LIN {X 0,Y 566.722,Z 306.411,A -85,B 0,C 180,E1 -2622.534,E2 -2622.534} C_VEL
LIN {X 0,Y 565.899,Z 301.524,A -85,B 0,C 180,E1 -2622.643,E2 -2622.643} C_VEL
LIN {X 0,Y 565.948,Z 295.461,A -85,B 0,C 180,E1 -2625.116,E2 -2625.116} C_VEL
LIN {X 0,Y 565.984,Z 288.275,A -85,B 0,C 180,E1 -2628.085,E2 -2628.085} C_VEL
LIN {X 0,Y 566.059,Z 281.089,A -85,B 0,C 180,E1 -2631.103,E2 -2631.103} C_VEL
LIN {X 0,Y 566.08,Z 273.903,A -85,B 0,C 180,E1 -2634.186,E2 -2634.186} C_VEL
LIN {X 0,Y 566.13,Z 268.296,A -85,B 0,C 180,E1 -2636.641,E2 -2636.641} C_VEL
LIN {X 0,Y 566.201,Z 261.327,A -85,B 0,C 180,E1 -2639.768,E2 -2639.768} C_VEL
LIN {X 0,Y 566.246,Z 255.555,A -85,B 0,C 180,E1 -2642.434,E2 -2642.434} C_VEL
LIN {X 0,Y 566.295,Z 250.149,A -85,B 0,C 180,E1 -2645.004,E2 -2645.004} C_VEL
LIN {X 0,Y 566.408,Z 245.469,A -85,B 0,C 180,E1 -2647.444,E2 -2647.444} C_VEL
LIN {X 0,Y 566.539,Z 240.518,A -85,B 0,C 180,E1 -2650.17,E2 -2650.17} C_VEL
LIN {X 0,Y 566.466,Z 237.367,A -85,B 0,C 180,E1 -2652.063,E2 -2652.063} C_VEL
LIN {X 0,Y 566.201,Z 235.83,A -85,B 0,C 180,E1 -2653.053,E2 -2653.053} C_VEL
LIN {X 0,Y 566.162,Z 235.462,A -85,B 0,C 180,E1 -2654.038,E2 -2654.038} C_VEL
LIN {X 0,Y 566.185,Z 235.462,A -85,B 0,C 180,E1 -2657.083,E2 -2657.083} C_VEL
LIN {X 0,Y 566.209,Z 235.454,A -85,B 0,C 180,E1 -2660.314,E2 -2660.314} C_VEL
LIN {X 0,Y 566.182,Z 235.455,A -85,B 0,C 180,E1 -2663.426,E2 -2663.426} C_VEL
LIN {X 0,Y 566.199,Z 235.455,A -85,B 0,C 180,E1 -2666.266,E2 -2666.266} C_VEL
LIN {X 0,Y 566.186,Z 235.458,A -85,B 0,C 180,E1 -2668.923,E2 -2668.923} C_VEL
LIN {X 0,Y 566.15,Z 235.459,A -85,B 0,C 180,E1 -2671.851,E2 -2671.851} C_VEL
LIN {X 0,Y 566.193,Z 235.458,A -85,B 0,C 180,E1 -2674.247,E2 -2674.247} C_VEL
LIN {X 0,Y 566.161,Z 235.456,A -85,B 0,C 180,E1 -2677.365,E2 -2677.365} C_VEL
LIN {X 0,Y 566.17,Z 235.456,A -85,B 0,C 180,E1 -2679.658,E2 -2679.658} C_VEL
LIN {X 0,Y 566.166,Z 235.46,A -85,B 0,C 180,E1 -2681.917,E2 -2681.917} C_VEL
LIN {X 0,Y 566.182,Z 235.454,A -85,B 0,C 180,E1 -2684.887,E2 -2684.887} C_VEL
LIN {X 0,Y 566.21,Z 235.456,A -85,B 0,C 180,E1 -2687.815,E2 -2687.815} C_VEL
LIN {X 0,Y 566.16,Z 235.466,A -85,B 0,C 180,E1 -2689.988,E2 -2689.988} C_VEL
LIN {X 0,Y 566.185,Z 235.459,A -85,B 0,C 180,E1 -2692.149,E2 -2692.149} C_VEL
LIN {X 0,Y 566.256,Z 235.445,A -85,B 0,C 180,E1 -2695.012,E2 -2695.012} C_VEL
LIN {X 0,Y 566.262,Z 235.451,A -85,B 0,C 180,E1 -2697.862,E2 -2697.862} C_VEL
LIN {X 0,Y 566.269,Z 235.447,A -85,B 0,C 180,E1 -2699.996,E2 -2699.996} C_VEL
LIN {X 0,Y 566.244,Z 235.446,A -85,B 0,C 180,E1 -2702.841,E2 -2702.841} C_VEL
LIN {X 0,Y 566.236,Z 235.454,A -85,B 0,C 180,E1 -2705.694,E2 -2705.694} C_VEL
LIN {X 0,Y 566.177,Z 235.454,A -85,B 0,C 180,E1 -2708.562,E2 -2708.562} C_VEL
LIN {X 0,Y 566.226,Z 235.456,A -85,B 0,C 180,E1 -2711.45,E2 -2711.45} C_VEL
LIN {X 0,Y 566.184,Z 235.454,A -85,B 0,C 180,E1 -2714.49,E2 -2714.49} C_VEL
LIN {X 0,Y 566.173,Z 235.462,A -85,B 0,C 180,E1 -2717.327,E2 -2717.327} C_VEL
LIN {X 0,Y 566.179,Z 235.454,A -85,B 0,C 180,E1 -2720.333,E2 -2720.333} C_VEL
LIN {X 0,Y 566.141,Z 235.464,A -85,B 0,C 180,E1 -2723.277,E2 -2723.277} C_VEL
LIN {X 0,Y 566.176,Z 235.454,A -85,B 0,C 180,E1 -2725.745,E2 -2725.745} C_VEL
LIN {X 0,Y 566.174,Z 235.456,A -85,B 0,C 180,E1 -2727.443,E2 -2727.443} C_VEL
LIN {X 0,Y 565.499,Z 235.54,A -85,B 0,C 180,E1 -2728.037,E2 -2728.037} C_VEL
LIN {X 0,Y 562.633,Z 235.902,A -85,B 0,C 180,E1 -2729.001,E2 -2729.001} C_VEL
LIN {X 0,Y 560.217,Z 236.2,A -85,B 0,C 180,E1 -2729.776,E2 -2729.776} C_VEL
LIN {X 0,Y 559.185,Z 236.329,A -85,B 0,C 180,E1 -2730.375,E2 -2730.375} C_VEL
LIN {X 0,Y 559.103,Z 236.337,A -85,B 0,C 180,E1 -2730.578,E2 -2730.578} C_VEL
LIN {X 0,Y 559.116,Z 236.344,A -85,B 0,C 180,E1 -2732.711,E2 -2732.711} C_VEL
LIN {X 0,Y 559.118,Z 236.334,A -85,B 0,C 180,E1 -2735.317,E2 -2735.317} C_VEL
LIN {X 0,Y 559.09,Z 236.339,A -85,B 0,C 180,E1 -2738.013,E2 -2738.013} C_VEL
LIN {X 0,Y 559.13,Z 236.336,A -85,B 0,C 180,E1 -2740.806,E2 -2740.806} C_VEL
LIN {X 0,Y 559.116,Z 236.335,A -85,B 0,C 180,E1 -2743.727,E2 -2743.727} C_VEL
LIN {X 0,Y 559.115,Z 236.336,A -85,B 0,C 180,E1 -2746.797,E2 -2746.797} C_VEL
LIN {X 0,Y 559.127,Z 236.332,A -85,B 0,C 180,E1 -2749.186,E2 -2749.186} C_VEL
LIN {X 0,Y 559.082,Z 236.345,A -85,B 0,C 180,E1 -2751.979,E2 -2751.979} C_VEL
LIN {X 0,Y 559.103,Z 236.336,A -85,B 0,C 180,E1 -2754.779,E2 -2754.779} C_VEL
LIN {X 0,Y 559.117,Z 236.335,A -85,B 0,C 180,E1 -2757.358,E2 -2757.358} C_VEL
LIN {X 0,Y 559.139,Z 236.337,A -85,B 0,C 180,E1 -2760.13,E2 -2760.13} C_VEL
LIN {X 0,Y 559.121,Z 236.334,A -85,B 0,C 180,E1 -2763.167,E2 -2763.167} C_VEL
LIN {X 0,Y 559.111,Z 236.34,A -85,B 0,C 180,E1 -2765.493,E2 -2765.493} C_VEL
LIN {X 0,Y 559.104,Z 236.342,A -85,B 0,C 180,E1 -2767.846,E2 -2767.846} C_VEL
LIN {X 0,Y 559.131,Z 236.332,A -85,B 0,C 180,E1 -2770.49,E2 -2770.49} C_VEL
LIN {X 0,Y 559.147,Z 236.336,A -85,B 0,C 180,E1 -2773.197,E2 -2773.197} C_VEL
LIN {X 0,Y 559.122,Z 236.335,A -85,B 0,C 180,E1 -2776.183,E2 -2776.183} C_VEL
LIN {X 0,Y 559.171,Z 236.334,A -85,B 0,C 180,E1 -2779.133,E2 -2779.133} C_VEL
LIN {X 0,Y 559.15,Z 236.331,A -85,B 0,C 180,E1 -2782.053,E2 -2782.053} C_VEL
LIN {X 0,Y 559.203,Z 236.33,A -85,B 0,C 180,E1 -2784.953,E2 -2784.953} C_VEL
LIN {X 0,Y 559.183,Z 236.327,A -85,B 0,C 180,E1 -2787.839,E2 -2787.839} C_VEL
LIN {X 0,Y 559.219,Z 236.328,A -85,B 0,C 180,E1 -2790.72,E2 -2790.72} C_VEL
LIN {X 0,Y 559.188,Z 236.334,A -85,B 0,C 180,E1 -2792.882,E2 -2792.882} C_VEL
LIN {X 0,Y 559.172,Z 236.328,A -85,B 0,C 180,E1 -2795.771,E2 -2795.771} C_VEL
LIN {X 0,Y 559.15,Z 236.331,A -85,B 0,C 180,E1 -2797.947,E2 -2797.947} C_VEL
LIN {X 0,Y 559.171,Z 236.334,A -85,B 0,C 180,E1 -2800.867,E2 -2800.867} C_VEL
LIN {X 0,Y 559.122,Z 236.335,A -85,B 0,C 180,E1 -2803.817,E2 -2803.817} C_VEL
LIN {X 0,Y 559.147,Z 236.336,A -85,B 0,C 180,E1 -2806.803,E2 -2806.803} C_VEL
LIN {X 0,Y 559.113,Z 236.336,A -85,B 0,C 180,E1 -2809.839,E2 -2809.839} C_VEL
LIN {X 0,Y 559.104,Z 236.342,A -85,B 0,C 180,E1 -2812.154,E2 -2812.154} C_VEL
LIN {X 0,Y 559.111,Z 236.34,A -85,B 0,C 180,E1 -2814.507,E2 -2814.507} C_VEL
LIN {X 0,Y 559.118,Z 236.334,A -85,B 0,C 180,E1 -2816.904,E2 -2816.904} C_VEL
LIN {X 0,Y 559.139,Z 236.337,A -85,B 0,C 180,E1 -2819.87,E2 -2819.87} C_VEL
LIN {X 0,Y 559.118,Z 236.334,A -85,B 0,C 180,E1 -2822.717,E2 -2822.717} C_VEL
LIN {X 0,Y 559.102,Z 236.337,A -85,B 0,C 180,E1 -2825.325,E2 -2825.325} C_VEL
LIN {X 0,Y 559.082,Z 236.345,A -85,B 0,C 180,E1 -2828.021,E2 -2828.021} C_VEL
LIN {X 0,Y 559.127,Z 236.332,A -85,B 0,C 180,E1 -2830.814,E2 -2830.814} C_VEL
LIN {X 0,Y 559.111,Z 236.343,A -85,B 0,C 180,E1 -2833.736,E2 -2833.736} C_VEL
LIN {X 0,Y 559.126,Z 236.333,A -85,B 0,C 180,E1 -2836.805,E2 -2836.805} C_VEL
LIN {X 0,Y 559.13,Z 236.336,A -85,B 0,C 180,E1 -2839.194,E2 -2839.194} C_VEL
LIN {X 0,Y 559.09,Z 236.339,A -85,B 0,C 180,E1 -2841.987,E2 -2841.987} C_VEL
LIN {X 0,Y 559.119,Z 236.335,A -85,B 0,C 180,E1 -2844.788,E2 -2844.788} C_VEL
LIN {X 0,Y 559.117,Z 236.342,A -85,B 0,C 180,E1 -2847.369,E2 -2847.369} C_VEL
LIN {X 0,Y 559.113,Z 236.334,A -85,B 0,C 180,E1 -2850.147,E2 -2850.147} C_VEL
LIN {X 0,Y 559.138,Z 236.341,A -85,B 0,C 180,E1 -2853.103,E2 -2853.103} C_VEL
LIN {X 0,Y 559.124,Z 236.336,A -85,B 0,C 180,E1 -2855.5,E2 -2855.5} C_VEL
LIN {X 0,Y 559.144,Z 236.335,A -85,B 0,C 180,E1 -2858.629,E2 -2858.629} C_VEL
LIN {X 0,Y 559.134,Z 236.34,A -85,B 0,C 180,E1 -2860.931,E2 -2860.931} C_VEL
LIN {X 0,Y 559.137,Z 236.331,A -85,B 0,C 180,E1 -2863.952,E2 -2863.952} C_VEL
LIN {X 0,Y 559.133,Z 236.338,A -85,B 0,C 180,E1 -2866.929,E2 -2866.929} C_VEL
LIN {X 0,Y 559.177,Z 236.329,A -85,B 0,C 180,E1 -2869.138,E2 -2869.138} C_VEL
LIN {X 0,Y 559.173,Z 236.329,A -85,B 0,C 180,E1 -2872.058,E2 -2872.058} C_VEL
LIN {X 0,Y 559.226,Z 236.323,A -85,B 0,C 180,E1 -2874.958,E2 -2874.958} C_VEL
LIN {X 0,Y 559.228,Z 236.322,A -85,B 0,C 180,E1 -2877.844,E2 -2877.844} C_VEL
LIN {X 0,Y 559.259,Z 236.319,A -85,B 0,C 180,E1 -2880.724,E2 -2880.724} C_VEL
LIN {X 0,Y 559.213,Z 236.323,A -85,B 0,C 180,E1 -2882.886,E2 -2882.886} C_VEL
LIN {X 0,Y 559.198,Z 236.327,A -85,B 0,C 180,E1 -2885.774,E2 -2885.774} C_VEL
LIN {X 0,Y 559.157,Z 236.33,A -85,B 0,C 180,E1 -2888.679,E2 -2888.679} C_VEL
LIN {X 0,Y 559.198,Z 236.327,A -85,B 0,C 180,E1 -2891.604,E2 -2891.604} C_VEL
LIN {X 0,Y 559.18,Z 236.327,A -85,B 0,C 180,E1 -2894.591,E2 -2894.591} C_VEL
LIN {X 0,Y 559.11,Z 236.34,A -85,B 0,C 180,E1 -2897.562,E2 -2897.562} C_VEL
LIN {X 0,Y 559.154,Z 236.337,A -85,B 0,C 180,E1 -2899.841,E2 -2899.841} C_VEL
LIN {X 0,Y 559.13,Z 236.334,A -85,B 0,C 180,E1 -2902.156,E2 -2902.156} C_VEL
LIN {X 0,Y 559.141,Z 236.334,A -85,B 0,C 180,E1 -2905.181,E2 -2905.181} C_VEL
LIN {X 0,Y 559.106,Z 236.341,A -85,B 0,C 180,E1 -2907.719,E2 -2907.719} C_VEL
LIN {X 0,Y 559.137,Z 236.332,A -85,B 0,C 180,E1 -2910.187,E2 -2910.187} C_VEL
LIN {X 0,Y 559.15,Z 236.331,A -85,B 0,C 180,E1 -2912.718,E2 -2912.718} C_VEL
LIN {X 0,Y 559.12,Z 236.342,A -85,B 0,C 180,E1 -2915.327,E2 -2915.327} C_VEL
LIN {X 0,Y 559.127,Z 236.334,A -85,B 0,C 180,E1 -2918.021,E2 -2918.021} C_VEL
LIN {X 0,Y 559.157,Z 236.336,A -85,B 0,C 180,E1 -2920.815,E2 -2920.815} C_VEL
LIN {X 0,Y 559.111,Z 236.339,A -85,B 0,C 180,E1 -2923.739,E2 -2923.739} C_VEL
LIN {X 0,Y 559.119,Z 236.342,A -85,B 0,C 180,E1 -2926.265,E2 -2926.265} C_VEL
LIN {X 0,Y 559.534,Z 239.189,A -85,B 0,C 180,E1 -2928.265,E2 -2928.265} C_VEL
LIN {X 0,Y 559.517,Z 242.348,A -85,B 0,C 180,E1 -2930.164,E2 -2930.164} C_VEL
LIN {X 0,Y 559.377,Z 247.292,A -85,B 0,C 180,E1 -2932.911,E2 -2932.911} C_VEL
LIN {X 0,Y 559.249,Z 252.345,A -85,B 0,C 180,E1 -2935.563,E2 -2935.563} C_VEL
LIN {X 0,Y 559.202,Z 257.734,A -85,B 0,C 180,E1 -2938.14,E2 -2938.14} C_VEL
LIN {X 0,Y 559.128,Z 263.124,A -85,B 0,C 180,E1 -2940.646,E2 -2940.646} C_VEL
LIN {X 0,Y 559.095,Z 268.727,A -85,B 0,C 180,E1 -2943.19,E2 -2943.19} C_VEL
LIN {X 0,Y 559.025,Z 273.903,A -85,B 0,C 180,E1 -2945.489,E2 -2945.489} C_VEL
LIN {X 0,Y 559.001,Z 281.089,A -85,B 0,C 180,E1 -2948.617,E2 -2948.617} C_VEL
LIN {X 0,Y 558.931,Z 286.478,A -85,B 0,C 180,E1 -2950.918,E2 -2950.918} C_VEL
LIN {X 0,Y 558.884,Z 291.868,A -85,B 0,C 180,E1 -2953.189,E2 -2953.189} C_VEL
LIN {X 0,Y 558.843,Z 299.054,A -85,B 0,C 180,E1 -2956.176,E2 -2956.176} C_VEL
LIN {X 0,Y 558.835,Z 301.524,A -85,B 0,C 180,E1 -2957.194,E2 -2957.194} C_VEL
LIN {X 0,Y 559.967,Z 309.414,A -85,B 0,C 180,E1 -2957.382,E2 -2957.382} C_VEL
LIN {X 0,Y 559.851,Z 321.119,A -85,B 0,C 180,E1 -2957.724,E2 -2957.724} C_VEL
LIN {X 0,Y 559.715,Z 331.464,A -85,B 0,C 180,E1 -2958.135,E2 -2958.135} C_VEL
LIN {X 0,Y 559.551,Z 342.846,A -85,B 0,C 180,E1 -2958.72,E2 -2958.72} C_VEL
LIN {X 0,Y 559.433,Z 354.75,A -85,B 0,C 180,E1 -2959.505,E2 -2959.505} C_VEL
LIN {X 0,Y 559.296,Z 363.641,A -85,B 0,C 180,E1 -2960.233,E2 -2960.233} C_VEL
LIN {X 0,Y 559.133,Z 372.762,A -85,B 0,C 180,E1 -2961.143,E2 -2961.143} C_VEL
LIN {X 0,Y 559.055,Z 380.309,A -85,B 0,C 180,E1 -2962.052,E2 -2962.052} C_VEL
LIN {X 0,Y 558.927,Z 387.956,A -85,B 0,C 180,E1 -2963.176,E2 -2963.176} C_VEL
LIN {X 0,Y 558.929,Z 393.682,A -85,B 0,C 180,E1 -2964.227,E2 -2964.227} C_VEL
LIN {X 0,Y 558.827,Z 398.379,A -85,B 0,C 180,E1 -2965.311,E2 -2965.311} C_VEL
LIN {X 0,Y 558.837,Z 401.966,A -85,B 0,C 180,E1 -2966.395,E2 -2966.395} C_VEL
LIN {X 0,Y 558.8,Z 403.792,A -85,B 0,C 180,E1 -2967.116,E2 -2967.116} C_VEL
LIN {X 0,Y 558.745,Z 406.19,A -85,B 0,C 180,E1 -2968.559,E2 -2968.559} C_VEL
LIN {X 0,Y 558.741,Z 406.782,A -85,B 0,C 180,E1 -2969.279,E2 -2969.279} C_VEL
LIN {X 0,Y 558.741,Z 406.782,A -85,B 0,C 180,E1 -2970.721,E2 -2970.721} C_VEL
LIN {X 0,Y 558.745,Z 406.19,A -85,B 0,C 180,E1 -2971.441,E2 -2971.441} C_VEL
LIN {X 0,Y 558.8,Z 403.792,A -85,B 0,C 180,E1 -2972.884,E2 -2972.884} C_VEL
LIN {X 0,Y 558.845,Z 400.88,A -85,B 0,C 180,E1 -2973.966,E2 -2973.966} C_VEL
LIN {X 0,Y 558.798,Z 396.93,A -85,B 0,C 180,E1 -2975.051,E2 -2975.051} C_VEL
LIN {X 0,Y 558.911,Z 391.835,A -85,B 0,C 180,E1 -2976.136,E2 -2976.136} C_VEL
LIN {X 0,Y 558.977,Z 385.452,A -85,B 0,C 180,E1 -2977.223,E2 -2977.223} C_VEL
LIN {X 0,Y 559.098,Z 377.491,A -85,B 0,C 180,E1 -2978.312,E2 -2978.312} C_VEL
LIN {X 0,Y 559.183,Z 369.35,A -85,B 0,C 180,E1 -2979.221,E2 -2979.221} C_VEL
LIN {X 0,Y 559.336,Z 359.358,A -85,B 0,C 180,E1 -2980.131,E2 -2980.131} C_VEL
LIN {X 0,Y 559.46,Z 349.539,A -85,B 0,C 180,E1 -2980.861,E2 -2980.861} C_VEL
LIN {X 0,Y 559.612,Z 338.508,A -85,B 0,C 180,E1 -2981.523,E2 -2981.523} C_VEL
LIN {X 0,Y 559.811,Z 324.985,A -85,B 0,C 180,E1 -2982.139,E2 -2982.139} C_VEL
LIN {X 0,Y 559.957,Z 312.983,A -85,B 0,C 180,E1 -2982.527,E2 -2982.527} C_VEL
LIN {X 0,Y 559.764,Z 307.128,A -85,B 0,C 180,E1 -2982.678,E2 -2982.678} C_VEL
LIN {X 0,Y 558.835,Z 301.524,A -85,B 0,C 180,E1 -2982.806,E2 -2982.806} C_VEL
LIN {X 0,Y 558.862,Z 295.461,A -85,B 0,C 180,E1 -2985.312,E2 -2985.312} C_VEL
LIN {X 0,Y 558.904,Z 288.275,A -85,B 0,C 180,E1 -2988.322,E2 -2988.322} C_VEL
LIN {X 0,Y 558.949,Z 282.885,A -85,B 0,C 180,E1 -2990.613,E2 -2990.613} C_VEL
LIN {X 0,Y 559.027,Z 276.436,A -85,B 0,C 180,E1 -2993.399,E2 -2993.399} C_VEL
LIN {X 0,Y 559.071,Z 270.31,A -85,B 0,C 180,E1 -2996.102,E2 -2996.102} C_VEL
LIN {X 0,Y 559.115,Z 264.92,A -85,B 0,C 180,E1 -2998.532,E2 -2998.532} C_VEL
LIN {X 0,Y 559.185,Z 258.975,A -85,B 0,C 180,E1 -3001.277,E2 -3001.277} C_VEL
LIN {X 0,Y 559.253,Z 253.328,A -85,B 0,C 180,E1 -3003.96,E2 -3003.96} C_VEL
LIN {X 0,Y 559.359,Z 248.434,A -85,B 0,C 180,E1 -3006.472,E2 -3006.472} C_VEL
LIN {X 0,Y 559.482,Z 243.98,A -85,B 0,C 180,E1 -3008.908,E2 -3008.908} C_VEL
LIN {X 0,Y 559.591,Z 240.185,A -85,B 0,C 180,E1 -3011.099,E2 -3011.099} C_VEL
LIN {X 0,Y 559.181,Z 236.927,A -85,B 0,C 180,E1 -3013.198,E2 -3013.198} C_VEL
LIN {X 0,Y 559.115,Z 236.341,A -85,B 0,C 180,E1 -3013.735,E2 -3013.735} C_VEL
LIN {X 0,Y 559.111,Z 236.338,A -85,B 0,C 180,E1 -3016.261,E2 -3016.261} C_VEL
LIN {X 0,Y 559.119,Z 236.34,A -85,B 0,C 180,E1 -3019.182,E2 -3019.182} C_VEL
LIN {X 0,Y 559.171,Z 236.333,A -85,B 0,C 180,E1 -3021.191,E2 -3021.191} C_VEL
LIN {X 0,Y 559.12,Z 236.333,A -85,B 0,C 180,E1 -3023.785,E2 -3023.785} C_VEL
LIN {X 0,Y 559.148,Z 236.335,A -85,B 0,C 180,E1 -3026.421,E2 -3026.421} C_VEL
LIN {X 0,Y 559.151,Z 236.333,A -85,B 0,C 180,E1 -3028.978,E2 -3028.978} C_VEL
LIN {X 0,Y 559.112,Z 236.334,A -85,B 0,C 180,E1 -3031.628,E2 -3031.628} C_VEL
LIN {X 0,Y 559.13,Z 236.337,A -85,B 0,C 180,E1 -3034.697,E2 -3034.697} C_VEL
LIN {X 0,Y 559.112,Z 236.335,A -85,B 0,C 180,E1 -3037.063,E2 -3037.063} C_VEL
LIN {X 0,Y 559.149,Z 236.33,A -85,B 0,C 180,E1 -3039.391,E2 -3039.391} C_VEL
LIN {X 0,Y 559.116,Z 236.336,A -85,B 0,C 180,E1 -3041.681,E2 -3041.681} C_VEL
LIN {X 0,Y 559.13,Z 236.334,A -85,B 0,C 180,E1 -3044.691,E2 -3044.691} C_VEL
LIN {X 0,Y 559.169,Z 236.331,A -85,B 0,C 180,E1 -3047.659,E2 -3047.659} C_VEL
LIN {X 0,Y 559.122,Z 236.341,A -85,B 0,C 180,E1 -3049.861,E2 -3049.861} C_VEL
LIN {X 0,Y 559.138,Z 236.339,A -85,B 0,C 180,E1 -3052.049,E2 -3052.049} C_VEL
LIN {X 0,Y 559.23,Z 236.32,A -85,B 0,C 180,E1 -3054.949,E2 -3054.949} C_VEL
LIN {X 0,Y 559.234,Z 236.327,A -85,B 0,C 180,E1 -3057.835,E2 -3057.835} C_VEL
LIN {X 0,Y 559.238,Z 236.323,A -85,B 0,C 180,E1 -3059.996,E2 -3059.996} C_VEL
LIN {X 0,Y 559.212,Z 236.322,A -85,B 0,C 180,E1 -3062.877,E2 -3062.877} C_VEL
LIN {X 0,Y 559.203,Z 236.328,A -85,B 0,C 180,E1 -3065.766,E2 -3065.766} C_VEL
LIN {X 0,Y 559.143,Z 236.331,A -85,B 0,C 180,E1 -3068.67,E2 -3068.67} C_VEL
LIN {X 0,Y 559.187,Z 236.33,A -85,B 0,C 180,E1 -3071.596,E2 -3071.596} C_VEL
LIN {X 0,Y 559.133,Z 236.333,A -85,B 0,C 180,E1 -3074.573,E2 -3074.573} C_VEL
LIN {X 0,Y 559.147,Z 236.339,A -85,B 0,C 180,E1 -3077.208,E2 -3077.208} C_VEL
LIN {X 0,Y 559.139,Z 236.332,A -85,B 0,C 180,E1 -3079.833,E2 -3079.833} C_VEL
LIN {X 0,Y 559.112,Z 236.334,A -85,B 0,C 180,E1 -3082.148,E2 -3082.148} C_VEL
LIN {X 0,Y 559.144,Z 236.334,A -85,B 0,C 180,E1 -3085.293,E2 -3085.293} C_VEL
LIN {X 0,Y 559.155,Z 236.329,A -85,B 0,C 180,E1 -3087.707,E2 -3087.707} C_VEL
LIN {X 0,Y 559.103,Z 236.337,A -85,B 0,C 180,E1 -3090.578,E2 -3090.578} C_VEL
LIN {X 0,Y 558.439,Z 236.423,A -85,B 0,C 180,E1 -3091.179,E2 -3091.179} C_VEL
LIN {X 0,Y 555.575,Z 236.777,A -85,B 0,C 180,E1 -3092.155,E2 -3092.155} C_VEL
LIN {X 0,Y 553.164,Z 237.081,A -85,B 0,C 180,E1 -3092.941,E2 -3092.941} C_VEL
LIN {X 0,Y 552.145,Z 237.203,A -85,B 0,C 180,E1 -3093.548,E2 -3093.548} C_VEL
LIN {X 0,Y 552.071,Z 237.211,A -85,B 0,C 180,E1 -3093.753,E2 -3093.753} C_VEL
LIN {X 0,Y 552.07,Z 237.218,A -85,B 0,C 180,E1 -3096.742,E2 -3096.742} C_VEL
LIN {X 0,Y 552.087,Z 237.209,A -85,B 0,C 180,E1 -3099.522,E2 -3099.522} C_VEL
LIN {X 0,Y 552.085,Z 237.219,A -85,B 0,C 180,E1 -3102.421,E2 -3102.421} C_VEL
LIN {X 0,Y 552.048,Z 237.215,A -85,B 0,C 180,E1 -3105.559,E2 -3105.559} C_VEL
LIN {X 0,Y 552.092,Z 237.212,A -85,B 0,C 180,E1 -3108.672,E2 -3108.672} C_VEL
LIN {X 0,Y 552.067,Z 237.212,A -85,B 0,C 180,E1 -3111.408,E2 -3111.408} C_VEL
LIN {X 0,Y 552.051,Z 237.216,A -85,B 0,C 180,E1 -3114.552,E2 -3114.552} C_VEL
LIN {X 0,Y 552.072,Z 237.211,A -85,B 0,C 180,E1 -3117.147,E2 -3117.147} C_VEL
LIN {X 0,Y 552.095,Z 237.213,A -85,B 0,C 180,E1 -3120.235,E2 -3120.235} C_VEL
LIN {X 0,Y 552.085,Z 237.21,A -85,B 0,C 180,E1 -3122.995,E2 -3122.995} C_VEL
LIN {X 0,Y 552.075,Z 237.213,A -85,B 0,C 180,E1 -3125.16,E2 -3125.16} C_VEL
LIN {X 0,Y 552.065,Z 237.22,A -85,B 0,C 180,E1 -3127.548,E2 -3127.548} C_VEL
LIN {X 0,Y 552.093,Z 237.209,A -85,B 0,C 180,E1 -3130.673,E2 -3130.673} C_VEL
LIN {X 0,Y 552.126,Z 237.208,A -85,B 0,C 180,E1 -3132.977,E2 -3132.977} C_VEL
LIN {X 0,Y 552.079,Z 237.213,A -85,B 0,C 180,E1 -3136.003,E2 -3136.003} C_VEL
LIN {X 0,Y 552.13,Z 237.209,A -85,B 0,C 180,E1 -3138.993,E2 -3138.993} C_VEL
LIN {X 0,Y 552.103,Z 237.21,A -85,B 0,C 180,E1 -3141.951,E2 -3141.951} C_VEL
LIN {X 0,Y 552.143,Z 237.204,A -85,B 0,C 180,E1 -3144.156,E2 -3144.156} C_VEL
LIN {X 0,Y 552.153,Z 237.21,A -85,B 0,C 180,E1 -3147.082,E2 -3147.082} C_VEL
LIN {X 0,Y 552.159,Z 237.202,A -85,B 0,C 180,E1 -3150,E2 -3150} C_VEL
LIN {X 0,Y 552.153,Z 237.21,A -85,B 0,C 180,E1 -3152.918,E2 -3152.918} C_VEL
LIN {X 0,Y 552.143,Z 237.204,A -85,B 0,C 180,E1 -3155.844,E2 -3155.844} C_VEL
LIN {X 0,Y 552.103,Z 237.21,A -85,B 0,C 180,E1 -3158.049,E2 -3158.049} C_VEL
LIN {X 0,Y 552.13,Z 237.209,A -85,B 0,C 180,E1 -3161.007,E2 -3161.007} C_VEL
LIN {X 0,Y 552.079,Z 237.213,A -85,B 0,C 180,E1 -3163.997,E2 -3163.997} C_VEL
LIN {X 0,Y 552.126,Z 237.206,A -85,B 0,C 180,E1 -3167.343,E2 -3167.343} C_VEL
LIN {X 0,Y 552.073,Z 237.216,A -85,B 0,C 180,E1 -3170.103,E2 -3170.103} C_VEL
LIN {X 0,Y 552.092,Z 237.209,A -85,B 0,C 180,E1 -3173.242,E2 -3173.242} C_VEL
LIN {X 0,Y 552.111,Z 237.208,A -85,B 0,C 180,E1 -3175.645,E2 -3175.645} C_VEL
LIN {X 0,Y 552.074,Z 237.214,A -85,B 0,C 180,E1 -3178.567,E2 -3178.567} C_VEL
LIN {X 0,Y 552.075,Z 237.213,A -85,B 0,C 180,E1 -3181.483,E2 -3181.483} C_VEL
LIN {X 0,Y 552.089,Z 237.215,A -85,B 0,C 180,E1 -3184.176,E2 -3184.176} C_VEL
LIN {X 0,Y 552.056,Z 237.213,A -85,B 0,C 180,E1 -3186.75,E2 -3186.75} C_VEL
LIN {X 0,Y 552.083,Z 237.215,A -85,B 0,C 180,E1 -3189.53,E2 -3189.53} C_VEL
LIN {X 0,Y 552.079,Z 237.211,A -85,B 0,C 180,E1 -3192.429,E2 -3192.429} C_VEL
LIN {X 0,Y 552.05,Z 237.222,A -85,B 0,C 180,E1 -3195.567,E2 -3195.567} C_VEL
LIN {X 0,Y 552.095,Z 237.209,A -85,B 0,C 180,E1 -3198.68,E2 -3198.68} C_VEL
LIN {X 0,Y 552.074,Z 237.22,A -85,B 0,C 180,E1 -3201.416,E2 -3201.416} C_VEL
LIN {X 0,Y 552.073,Z 237.212,A -85,B 0,C 180,E1 -3204.163,E2 -3204.163} C_VEL
LIN {X 0,Y 552.075,Z 237.213,A -85,B 0,C 180,E1 -3206.819,E2 -3206.819} C_VEL
LIN {X 0,Y 552.066,Z 237.219,A -85,B 0,C 180,E1 -3209.396,E2 -3209.396} C_VEL
LIN {X 0,Y 552.092,Z 237.209,A -85,B 0,C 180,E1 -3211.907,E2 -3211.907} C_VEL
LIN {X 0,Y 552.106,Z 237.21,A -85,B 0,C 180,E1 -3214.659,E2 -3214.659} C_VEL
LIN {X 0,Y 552.063,Z 237.214,A -85,B 0,C 180,E1 -3217.554,E2 -3217.554} C_VEL
LIN {X 0,Y 552.118,Z 237.208,A -85,B 0,C 180,E1 -3220.38,E2 -3220.38} C_VEL
LIN {X 0,Y 552.109,Z 237.214,A -85,B 0,C 180,E1 -3222.981,E2 -3222.981} C_VEL
LIN {X 0,Y 552.089,Z 237.21,A -85,B 0,C 180,E1 -3226.009,E2 -3226.009} C_VEL
LIN {X 0,Y 552.146,Z 237.206,A -85,B 0,C 180,E1 -3228.998,E2 -3228.998} C_VEL
LIN {X 0,Y 552.128,Z 237.206,A -85,B 0,C 180,E1 -3231.956,E2 -3231.956} C_VEL
LIN {X 0,Y 552.202,Z 237.198,A -85,B 0,C 180,E1 -3234.893,E2 -3234.893} C_VEL
LIN {X 0,Y 552.2,Z 237.197,A -85,B 0,C 180,E1 -3237.816,E2 -3237.816} C_VEL
LIN {X 0,Y 552.229,Z 237.195,A -85,B 0,C 180,E1 -3240.733,E2 -3240.733} C_VEL
LIN {X 0,Y 552.179,Z 237.199,A -85,B 0,C 180,E1 -3242.922,E2 -3242.922} C_VEL
LIN {X 0,Y 552.17,Z 237.204,A -85,B 0,C 180,E1 -3245.848,E2 -3245.848} C_VEL
LIN {X 0,Y 552.128,Z 237.205,A -85,B 0,C 180,E1 -3248.79,E2 -3248.79} C_VEL
LIN {X 0,Y 552.155,Z 237.207,A -85,B 0,C 180,E1 -3251.754,E2 -3251.754} C_VEL
LIN {X 0,Y 552.127,Z 237.204,A -85,B 0,C 180,E1 -3254.752,E2 -3254.752} C_VEL
LIN {X 0,Y 552.076,Z 237.22,A -85,B 0,C 180,E1 -3257.793,E2 -3257.793} C_VEL
LIN {X 0,Y 552.112,Z 237.21,A -85,B 0,C 180,E1 -3260.105,E2 -3260.105} C_VEL
LIN {X 0,Y 552.083,Z 237.21,A -85,B 0,C 180,E1 -3262.455,E2 -3262.455} C_VEL
LIN {X 0,Y 552.086,Z 237.215,A -85,B 0,C 180,E1 -3265.337,E2 -3265.337} C_VEL
LIN {X 0,Y 552.056,Z 237.215,A -85,B 0,C 180,E1 -3268.104,E2 -3268.104} C_VEL
LIN {X 0,Y 552.094,Z 237.209,A -85,B 0,C 180,E1 -3270.613,E2 -3270.613} C_VEL
LIN {X 0,Y 552.107,Z 237.214,A -85,B 0,C 180,E1 -3273.189,E2 -3273.189} C_VEL
LIN {X 0,Y 552.074,Z 237.214,A -85,B 0,C 180,E1 -3275.847,E2 -3275.847} C_VEL
LIN {X 0,Y 552.114,Z 237.21,A -85,B 0,C 180,E1 -3278.592,E2 -3278.592} C_VEL
LIN {X 0,Y 552.071,Z 237.218,A -85,B 0,C 180,E1 -3281.453,E2 -3281.453} C_VEL
LIN {X 0,Y 552.08,Z 237.218,A -85,B 0,C 180,E1 -3284.531,E2 -3284.531} C_VEL
LIN {X 0,Y 552.079,Z 237.218,A -85,B 0,C 180,E1 -3285.562,E2 -3285.562} C_VEL
LIN {X 0,Y 552.168,Z 237.905,A -85,B 0,C 180,E1 -3286.583,E2 -3286.583} C_VEL
LIN {X 0,Y 552.573,Z 241.048,A -85,B 0,C 180,E1 -3288.628,E2 -3288.628} C_VEL
LIN {X 0,Y 552.465,Z 245.792,A -85,B 0,C 180,E1 -3291.441,E2 -3291.441} C_VEL
LIN {X 0,Y 552.281,Z 251.439,A -85,B 0,C 180,E1 -3294.533,E2 -3294.533} C_VEL
LIN {X 0,Y 552.202,Z 256.601,A -85,B 0,C 180,E1 -3297.142,E2 -3297.142} C_VEL
LIN {X 0,Y 552.122,Z 262.514,A -85,B 0,C 180,E1 -3299.951,E2 -3299.951} C_VEL
LIN {X 0,Y 552.049,Z 269.167,A -85,B 0,C 180,E1 -3303.021,E2 -3303.021} C_VEL
LIN {X 0,Y 551.954,Z 275.699,A -85,B 0,C 180,E1 -3305.955,E2 -3305.955} C_VEL
LIN {X 0,Y 551.949,Z 281.16,A -85,B 0,C 180,E1 -3308.362,E2 -3308.362} C_VEL
LIN {X 0,Y 551.866,Z 286.478,A -85,B 0,C 180,E1 -3310.664,E2 -3310.664} C_VEL
LIN {X 0,Y 551.825,Z 291.868,A -85,B 0,C 180,E1 -3312.967,E2 -3312.967} C_VEL
LIN {X 0,Y 551.759,Z 299.054,A -85,B 0,C 180,E1 -3315.995,E2 -3315.995} C_VEL
LIN {X 0,Y 551.732,Z 301.524,A -85,B 0,C 180,E1 -3317.026,E2 -3317.026} C_VEL
LIN {X 0,Y 553.045,Z 310.323,A -85,B 0,C 180,E1 -3317.244,E2 -3317.244} C_VEL
LIN {X 0,Y 552.9,Z 322.4,A -85,B 0,C 180,E1 -3317.614,E2 -3317.614} C_VEL
LIN {X 0,Y 552.745,Z 333.449,A -85,B 0,C 180,E1 -3318.076,E2 -3318.076} C_VEL
LIN {X 0,Y 552.578,Z 345.38,A -85,B 0,C 180,E1 -3318.726,E2 -3318.726} C_VEL
LIN {X 0,Y 552.385,Z 357.081,A -85,B 0,C 180,E1 -3319.555,E2 -3319.555} C_VEL
LIN {X 0,Y 552.232,Z 365.578,A -85,B 0,C 180,E1 -3320.292,E2 -3320.292} C_VEL
LIN {X 0,Y 552.078,Z 374.381,A -85,B 0,C 180,E1 -3321.213,E2 -3321.213} C_VEL
LIN {X 0,Y 551.952,Z 383.009,A -85,B 0,C 180,E1 -3322.317,E2 -3322.317} C_VEL
LIN {X 0,Y 551.828,Z 389.873,A -85,B 0,C 180,E1 -3323.418,E2 -3323.418} C_VEL
LIN {X 0,Y 551.802,Z 395.364,A -85,B 0,C 180,E1 -3324.519,E2 -3324.519} C_VEL
LIN {X 0,Y 551.765,Z 399.663,A -85,B 0,C 180,E1 -3325.617,E2 -3325.617} C_VEL
LIN {X 0,Y 551.751,Z 401.967,A -85,B 0,C 180,E1 -3326.349,E2 -3326.349} C_VEL
LIN {X 0,Y 551.725,Z 403.79,A -85,B 0,C 180,E1 -3327.079,E2 -3327.079} C_VEL
LIN {X 0,Y 551.645,Z 406.19,A -85,B 0,C 180,E1 -3328.54,E2 -3328.54} C_VEL
LIN {X 0,Y 551.641,Z 406.782,A -85,B 0,C 180,E1 -3329.27,E2 -3329.27} C_VEL
LIN {X 0,Y 551.641,Z 406.782,A -85,B 0,C 180,E1 -3330.73,E2 -3330.73} C_VEL
LIN {X 0,Y 551.645,Z 406.19,A -85,B 0,C 180,E1 -3331.46,E2 -3331.46} C_VEL
LIN {X 0,Y 551.725,Z 403.79,A -85,B 0,C 180,E1 -3332.921,E2 -3332.921} C_VEL
LIN {X 0,Y 551.765,Z 400.876,A -85,B 0,C 180,E1 -3334.017,E2 -3334.017} C_VEL
LIN {X 0,Y 551.724,Z 396.926,A -85,B 0,C 180,E1 -3335.116,E2 -3335.116} C_VEL
LIN {X 0,Y 551.838,Z 392.439,A -85,B 0,C 180,E1 -3336.097,E2 -3336.097} C_VEL
LIN {X 0,Y 551.89,Z 386.597,A -85,B 0,C 180,E1 -3337.132,E2 -3337.132} C_VEL
LIN {X 0,Y 552.014,Z 378.935,A -85,B 0,C 180,E1 -3338.235,E2 -3338.235} C_VEL
LIN {X 0,Y 552.157,Z 369.351,A -85,B 0,C 180,E1 -3339.339,E2 -3339.339} C_VEL
LIN {X 0,Y 552.334,Z 359.352,A -85,B 0,C 180,E1 -3340.261,E2 -3340.261} C_VEL
LIN {X 0,Y 552.483,Z 349.531,A -85,B 0,C 180,E1 -3341,E2 -3341} C_VEL
LIN {X 0,Y 552.666,Z 337.75,A -85,B 0,C 180,E1 -3341.71,E2 -3341.71} C_VEL
LIN {X 0,Y 552.87,Z 324.972,A -85,B 0,C 180,E1 -3342.293,E2 -3342.293} C_VEL
LIN {X 0,Y 553.038,Z 312.967,A -85,B 0,C 180,E1 -3342.686,E2 -3342.686} C_VEL
LIN {X 0,Y 552.824,Z 307.976,A -85,B 0,C 180,E1 -3342.821,E2 -3342.821} C_VEL
LIN {X 0,Y 551.732,Z 301.524,A -85,B 0,C 180,E1 -3342.974,E2 -3342.974} C_VEL
LIN {X 0,Y 551.776,Z 295.461,A -85,B 0,C 180,E1 -3345.514,E2 -3345.514} C_VEL
LIN {X 0,Y 551.827,Z 290.071,A -85,B 0,C 180,E1 -3347.798,E2 -3347.798} C_VEL
LIN {X 0,Y 551.895,Z 284.682,A -85,B 0,C 180,E1 -3350.11,E2 -3350.11} C_VEL
LIN {X 0,Y 551.918,Z 279.292,A -85,B 0,C 180,E1 -3352.458,E2 -3352.458} C_VEL
LIN {X 0,Y 552.002,Z 272.854,A -85,B 0,C 180,E1 -3355.314,E2 -3355.314} C_VEL
LIN {X 0,Y 552.047,Z 266.717,A -85,B 0,C 180,E1 -3358.101,E2 -3358.101} C_VEL
LIN {X 0,Y 552.118,Z 261.327,A -85,B 0,C 180,E1 -3360.608,E2 -3360.608} C_VEL
LIN {X 0,Y 552.206,Z 255.938,A -85,B 0,C 180,E1 -3363.179,E2 -3363.179} C_VEL
LIN {X 0,Y 552.303,Z 250.769,A -85,B 0,C 180,E1 -3365.827,E2 -3365.827} C_VEL
LIN {X 0,Y 552.465,Z 245.792,A -85,B 0,C 180,E1 -3368.559,E2 -3368.559} C_VEL
LIN {X 0,Y 552.57,Z 240.962,A -85,B 0,C 180,E1 -3371.404,E2 -3371.404} C_VEL
LIN {X 0,Y 552.16,Z 237.799,A -85,B 0,C 180,E1 -3373.487,E2 -3373.487} C_VEL
LIN {X 0,Y 552.079,Z 237.217,A -85,B 0,C 180,E1 -3374.528,E2 -3374.528} C_VEL
LIN {X 0,Y 552.088,Z 237.213,A -85,B 0,C 180,E1 -3377.588,E2 -3377.588} C_VEL
LIN {X 0,Y 552.126,Z 237.21,A -85,B 0,C 180,E1 -3380.47,E2 -3380.47} C_VEL
LIN {X 0,Y 552.102,Z 237.21,A -85,B 0,C 180,E1 -3383.316,E2 -3383.316} C_VEL
LIN {X 0,Y 552.1,Z 237.208,A -85,B 0,C 180,E1 -3385.934,E2 -3385.934} C_VEL
LIN {X 0,Y 552.108,Z 237.215,A -85,B 0,C 180,E1 -3388.537,E2 -3388.537} C_VEL
LIN {X 0,Y 552.081,Z 237.21,A -85,B 0,C 180,E1 -3391.445,E2 -3391.445} C_VEL
LIN {X 0,Y 552.084,Z 237.218,A -85,B 0,C 180,E1 -3394.35,E2 -3394.35} C_VEL
LIN {X 0,Y 552.09,Z 237.213,A -85,B 0,C 180,E1 -3396.754,E2 -3396.754} C_VEL
LIN {X 0,Y 552.097,Z 237.208,A -85,B 0,C 180,E1 -3399.116,E2 -3399.116} C_VEL
LIN {X 0,Y 552.079,Z 237.211,A -85,B 0,C 180,E1 -3401.439,E2 -3401.439} C_VEL
LIN {X 0,Y 552.087,Z 237.214,A -85,B 0,C 180,E1 -3404.491,E2 -3404.491} C_VEL
LIN {X 0,Y 552.109,Z 237.208,A -85,B 0,C 180,E1 -3406.751,E2 -3406.751} C_VEL
LIN {X 0,Y 552.156,Z 237.201,A -85,B 0,C 180,E1 -3408.99,E2 -3408.99} C_VEL
LIN {X 0,Y 552.107,Z 237.216,A -85,B 0,C 180,E1 -3411.947,E2 -3411.947} C_VEL
LIN {X 0,Y 552.206,Z 237.195,A -85,B 0,C 180,E1 -3414.885,E2 -3414.885} C_VEL
LIN {X 0,Y 552.206,Z 237.203,A -85,B 0,C 180,E1 -3417.808,E2 -3417.808} C_VEL
LIN {X 0,Y 552.208,Z 237.199,A -85,B 0,C 180,E1 -3419.996,E2 -3419.996} C_VEL
LIN {X 0,Y 552.181,Z 237.199,A -85,B 0,C 180,E1 -3422.914,E2 -3422.914} C_VEL
LIN {X 0,Y 552.171,Z 237.203,A -85,B 0,C 180,E1 -3425.84,E2 -3425.84} C_VEL
LIN {X 0,Y 552.116,Z 237.207,A -85,B 0,C 180,E1 -3428.782,E2 -3428.782} C_VEL
LIN {X 0,Y 552.143,Z 237.206,A -85,B 0,C 180,E1 -3431.746,E2 -3431.746} C_VEL
LIN {X 0,Y 552.099,Z 237.21,A -85,B 0,C 180,E1 -3434.744,E2 -3434.744} C_VEL
LIN {X 0,Y 552.073,Z 237.212,A -85,B 0,C 180,E1 -3437.784,E2 -3437.784} C_VEL
LIN {X 0,Y 552.099,Z 237.208,A -85,B 0,C 180,E1 -3440.097,E2 -3440.097} C_VEL
LIN {X 0,Y 552.063,Z 237.214,A -85,B 0,C 180,E1 -3442.446,E2 -3442.446} C_VEL
LIN {X 0,Y 552.106,Z 237.21,A -85,B 0,C 180,E1 -3445.341,E2 -3445.341} C_VEL
LIN {X 0,Y 552.089,Z 237.21,A -85,B 0,C 180,E1 -3448.093,E2 -3448.093} C_VEL
LIN {X 0,Y 552.066,Z 237.219,A -85,B 0,C 180,E1 -3450.604,E2 -3450.604} C_VEL
LIN {X 0,Y 552.075,Z 237.213,A -85,B 0,C 180,E1 -3453.181,E2 -3453.181} C_VEL
LIN {X 0,Y 552.071,Z 237.211,A -85,B 0,C 180,E1 -3453.753,E2 -3453.753} C_VEL
LIN {X 0,Y 551.438,Z 237.296,A -85,B 0,C 180,E1 -3454.362,E2 -3454.362} C_VEL
LIN {X 0,Y 548.622,Z 237.649,A -85,B 0,C 180,E1 -3455.35,E2 -3455.35} C_VEL
LIN {X 0,Y 546.203,Z 237.952,A -85,B 0,C 180,E1 -3456.146,E2 -3456.146} C_VEL
LIN {X 0,Y 545.131,Z 238.083,A -85,B 0,C 180,E1 -3456.76,E2 -3456.76} C_VEL
LIN {X 0,Y 545.027,Z 238.092,A -85,B 0,C 180,E1 -3456.968,E2 -3456.968} C_VEL
LIN {X 0,Y 545.027,Z 238.093,A -85,B 0,C 180,E1 -3460.137,E2 -3460.137} C_VEL
LIN {X 0,Y 545.042,Z 238.088,A -85,B 0,C 180,E1 -3463.101,E2 -3463.101} C_VEL
LIN {X 0,Y 545.013,Z 238.099,A -85,B 0,C 180,E1 -3466.22,E2 -3466.22} C_VEL
LIN {X 0,Y 545.052,Z 238.087,A -85,B 0,C 180,E1 -3468.884,E2 -3468.884} C_VEL
LIN {X 0,Y 545.001,Z 238.096,A -85,B 0,C 180,E1 -3471.759,E2 -3471.759} C_VEL
LIN {X 0,Y 545.009,Z 238.094,A -85,B 0,C 180,E1 -3474.53,E2 -3474.53} C_VEL
LIN {X 0,Y 545.025,Z 238.09,A -85,B 0,C 180,E1 -3477.209,E2 -3477.209} C_VEL
LIN {X 0,Y 545.041,Z 238.095,A -85,B 0,C 180,E1 -3479.81,E2 -3479.81} C_VEL
LIN {X 0,Y 545.04,Z 238.087,A -85,B 0,C 180,E1 -3482.822,E2 -3482.822} C_VEL
LIN {X 0,Y 545.018,Z 238.098,A -85,B 0,C 180,E1 -3485.63,E2 -3485.63} C_VEL
LIN {X 0,Y 545.034,Z 238.09,A -85,B 0,C 180,E1 -3488.168,E2 -3488.168} C_VEL
LIN {X 0,Y 545.025,Z 238.093,A -85,B 0,C 180,E1 -3491.194,E2 -3491.194} C_VEL
LIN {X 0,Y 545.037,Z 238.097,A -85,B 0,C 180,E1 -3493.52,E2 -3493.52} C_VEL
LIN {X 0,Y 545.034,Z 238.093,A -85,B 0,C 180,E1 -3495.819,E2 -3495.819} C_VEL
LIN {X 0,Y 545.078,Z 238.086,A -85,B 0,C 180,E1 -3498.849,E2 -3498.849} C_VEL
LIN {X 0,Y 545.073,Z 238.086,A -85,B 0,C 180,E1 -3501.846,E2 -3501.846} C_VEL
LIN {X 0,Y 545.115,Z 238.079,A -85,B 0,C 180,E1 -3504.08,E2 -3504.08} C_VEL
LIN {X 0,Y 545.118,Z 238.086,A -85,B 0,C 180,E1 -3507.044,E2 -3507.044} C_VEL
LIN {X 0,Y 545.129,Z 238.078,A -85,B 0,C 180,E1 -3510,E2 -3510} C_VEL
LIN {X 0,Y 545.118,Z 238.086,A -85,B 0,C 180,E1 -3512.956,E2 -3512.956} C_VEL
LIN {X 0,Y 545.115,Z 238.079,A -85,B 0,C 180,E1 -3515.92,E2 -3515.92} C_VEL
LIN {X 0,Y 545.073,Z 238.086,A -85,B 0,C 180,E1 -3518.154,E2 -3518.154} C_VEL
LIN {X 0,Y 545.078,Z 238.086,A -85,B 0,C 180,E1 -3521.151,E2 -3521.151} C_VEL
LIN {X 0,Y 545.034,Z 238.093,A -85,B 0,C 180,E1 -3524.181,E2 -3524.181} C_VEL
LIN {X 0,Y 545.074,Z 238.084,A -85,B 0,C 180,E1 -3527.447,E2 -3527.447} C_VEL
LIN {X 0,Y 545.037,Z 238.097,A -85,B 0,C 180,E1 -3530.374,E2 -3530.374} C_VEL
LIN {X 0,Y 545.087,Z 238.082,A -85,B 0,C 180,E1 -3533.559,E2 -3533.559} C_VEL
LIN {X 0,Y 545.044,Z 238.093,A -85,B 0,C 180,E1 -3536.002,E2 -3536.002} C_VEL
LIN {X 0,Y 545.039,Z 238.089,A -85,B 0,C 180,E1 -3538.754,E2 -3538.754} C_VEL
LIN {X 0,Y 545.02,Z 238.094,A -85,B 0,C 180,E1 -3541.686,E2 -3541.686} C_VEL
LIN {X 0,Y 545.028,Z 238.09,A -85,B 0,C 180,E1 -3544.566,E2 -3544.566} C_VEL
LIN {X 0,Y 544.985,Z 238.096,A -85,B 0,C 180,E1 -3547.307,E2 -3547.307} C_VEL
LIN {X 0,Y 545.042,Z 238.091,A -85,B 0,C 180,E1 -3550.144,E2 -3550.144} C_VEL
LIN {X 0,Y 545.035,Z 238.089,A -85,B 0,C 180,E1 -3553.11,E2 -3553.11} C_VEL
LIN {X 0,Y 545.019,Z 238.091,A -85,B 0,C 180,E1 -3556.229,E2 -3556.229} C_VEL
LIN {X 0,Y 545.055,Z 238.086,A -85,B 0,C 180,E1 -3558.892,E2 -3558.892} C_VEL
LIN {X 0,Y 545.009,Z 238.096,A -85,B 0,C 180,E1 -3561.767,E2 -3561.767} C_VEL
LIN {X 0,Y 545.025,Z 238.089,A -85,B 0,C 180,E1 -3564.538,E2 -3564.538} C_VEL
LIN {X 0,Y 545.029,Z 238.097,A -85,B 0,C 180,E1 -3567.216,E2 -3567.216} C_VEL
LIN {X 0,Y 545.028,Z 238.09,A -85,B 0,C 180,E1 -3569.815,E2 -3569.815} C_VEL
LIN {X 0,Y 545.06,Z 238.085,A -85,B 0,C 180,E1 -3572.349,E2 -3572.349} C_VEL
LIN {X 0,Y 545.074,Z 238.089,A -85,B 0,C 180,E1 -3574.825,E2 -3574.825} C_VEL
LIN {X 0,Y 545.008,Z 238.097,A -85,B 0,C 180,E1 -3577.247,E2 -3577.247} C_VEL
LIN {X 0,Y 545.09,Z 238.084,A -85,B 0,C 180,E1 -3580.42,E2 -3580.42} C_VEL
LIN {X 0,Y 545.039,Z 238.088,A -85,B 0,C 180,E1 -3583.526,E2 -3583.526} C_VEL
LIN {X 0,Y 545.047,Z 238.086,A -85,B 0,C 180,E1 -3585.824,E2 -3585.824} C_VEL
LIN {X 0,Y 545.101,Z 238.086,A -85,B 0,C 180,E1 -3588.854,E2 -3588.854} C_VEL
LIN {X 0,Y 545.076,Z 238.084,A -85,B 0,C 180,E1 -3591.851,E2 -3591.851} C_VEL
LIN {X 0,Y 545.178,Z 238.074,A -85,B 0,C 180,E1 -3594.827,E2 -3594.827} C_VEL
LIN {X 0,Y 545.173,Z 238.072,A -85,B 0,C 180,E1 -3597.788,E2 -3597.788} C_VEL
LIN {X 0,Y 545.199,Z 238.07,A -85,B 0,C 180,E1 -3600.743,E2 -3600.743} C_VEL
LIN {X 0,Y 545.145,Z 238.075,A -85,B 0,C 180,E1 -3602.96,E2 -3602.96} C_VEL
LIN {X 0,Y 545.12,Z 238.083,A -85,B 0,C 180,E1 -3605.924,E2 -3605.924} C_VEL
LIN {X 0,Y 545.089,Z 238.081,A -85,B 0,C 180,E1 -3608.904,E2 -3608.904} C_VEL
LIN {X 0,Y 545.098,Z 238.089,A -85,B 0,C 180,E1 -3611.909,E2 -3611.909} C_VEL
LIN {X 0,Y 545.078,Z 238.082,A -85,B 0,C 180,E1 -3614.947,E2 -3614.947} C_VEL
LIN {X 0,Y 545.046,Z 238.092,A -85,B 0,C 180,E1 -3618.03,E2 -3618.03} C_VEL
LIN {X 0,Y 545.05,Z 238.087,A -85,B 0,C 180,E1 -3620.377,E2 -3620.377} C_VEL
LIN {X 0,Y 545.028,Z 238.089,A -85,B 0,C 180,E1 -3622.761,E2 -3622.761} C_VEL
LIN {X 0,Y 545.038,Z 238.096,A -85,B 0,C 180,E1 -3625.498,E2 -3625.498} C_VEL
LIN {X 0,Y 545.041,Z 238.087,A -85,B 0,C 180,E1 -3628.499,E2 -3628.499} C_VEL
LIN {X 0,Y 545.057,Z 238.089,A -85,B 0,C 180,E1 -3631.051,E2 -3631.051} C_VEL
LIN {X 0,Y 545.049,Z 238.091,A -85,B 0,C 180,E1 -3633.676,E2 -3633.676} C_VEL
LIN {X 0,Y 545.068,Z 238.09,A -85,B 0,C 180,E1 -3636.927,E2 -3636.927} C_VEL
LIN {X 0,Y 545.066,Z 238.087,A -85,B 0,C 180,E1 -3640.145,E2 -3640.145} C_VEL
LIN {X 0,Y 545.023,Z 238.099,A -85,B 0,C 180,E1 -3643.115,E2 -3643.115} C_VEL
LIN {X 0,Y 545.028,Z 238.169,A -85,B 0,C 180,E1 -3645.869,E2 -3645.869} C_VEL
LIN {X 0,Y 545.542,Z 241.865,A -85,B 0,C 180,E1 -3648.35,E2 -3648.35} C_VEL
LIN {X 0,Y 545.529,Z 245.999,A -85,B 0,C 180,E1 -3650.858,E2 -3650.858} C_VEL
LIN {X 0,Y 545.309,Z 250.922,A -85,B 0,C 180,E1 -3653.641,E2 -3653.641} C_VEL
LIN {X 0,Y 545.194,Z 255.998,A -85,B 0,C 180,E1 -3656.338,E2 -3656.338} C_VEL
LIN {X 0,Y 545.094,Z 261.327,A -85,B 0,C 180,E1 -3658.955,E2 -3658.955} C_VEL
LIN {X 0,Y 545.028,Z 266.717,A -85,B 0,C 180,E1 -3661.504,E2 -3661.504} C_VEL
LIN {X 0,Y 544.95,Z 272.106,A -85,B 0,C 180,E1 -3663.993,E2 -3663.993} C_VEL
LIN {X 0,Y 544.878,Z 277.496,A -85,B 0,C 180,E1 -3666.432,E2 -3666.432} C_VEL
LIN {X 0,Y 544.849,Z 282.885,A -85,B 0,C 180,E1 -3668.828,E2 -3668.828} C_VEL
LIN {X 0,Y 544.753,Z 288.275,A -85,B 0,C 180,E1 -3671.184,E2 -3671.184} C_VEL
LIN {X 0,Y 544.711,Z 293.664,A -85,B 0,C 180,E1 -3673.51,E2 -3673.51} C_VEL
LIN {X 0,Y 544.691,Z 299.054,A -85,B 0,C 180,E1 -3675.809,E2 -3675.809} C_VEL
LIN {X 0,Y 544.634,Z 301.524,A -85,B 0,C 180,E1 -3676.854,E2 -3676.854} C_VEL
LIN {X 0,Y 546.13,Z 311.204,A -85,B 0,C 180,E1 -3677.104,E2 -3677.104} C_VEL
LIN {X 0,Y 545.962,Z 322.39,A -85,B 0,C 180,E1 -3677.454,E2 -3677.454} C_VEL
LIN {X 0,Y 545.788,Z 333.446,A -85,B 0,C 180,E1 -3677.922,E2 -3677.922} C_VEL
LIN {X 0,Y 545.585,Z 344.193,A -85,B 0,C 180,E1 -3678.508,E2 -3678.508} C_VEL
LIN {X 0,Y 545.391,Z 355.919,A -85,B 0,C 180,E1 -3679.325,E2 -3679.325} C_VEL
LIN {X 0,Y 545.226,Z 365.574,A -85,B 0,C 180,E1 -3680.166,E2 -3680.166} C_VEL
LIN {X 0,Y 545.051,Z 374.376,A -85,B 0,C 180,E1 -3681.099,E2 -3681.099} C_VEL
LIN {X 0,Y 544.899,Z 383.009,A -85,B 0,C 180,E1 -3682.217,E2 -3682.217} C_VEL
LIN {X 0,Y 544.765,Z 390.285,A -85,B 0,C 180,E1 -3683.408,E2 -3683.408} C_VEL
LIN {X 0,Y 544.739,Z 395.364,A -85,B 0,C 180,E1 -3684.447,E2 -3684.447} C_VEL
LIN {X 0,Y 544.661,Z 399.661,A -85,B 0,C 180,E1 -3685.56,E2 -3685.56} C_VEL
LIN {X 0,Y 544.67,Z 401.968,A -85,B 0,C 180,E1 -3686.301,E2 -3686.301} C_VEL
LIN {X 0,Y 544.652,Z 403.787,A -85,B 0,C 180,E1 -3687.041,E2 -3687.041} C_VEL
LIN {X 0,Y 544.546,Z 406.191,A -85,B 0,C 180,E1 -3688.521,E2 -3688.521} C_VEL
LIN {X 0,Y 544.542,Z 406.781,A -85,B 0,C 180,E1 -3689.261,E2 -3689.261} C_VEL
LIN {X 0,Y 544.542,Z 406.781,A -85,B 0,C 180,E1 -3690.739,E2 -3690.739} C_VEL
LIN {X 0,Y 544.546,Z 406.191,A -85,B 0,C 180,E1 -3691.479,E2 -3691.479} C_VEL
LIN {X 0,Y 544.652,Z 403.787,A -85,B 0,C 180,E1 -3692.959,E2 -3692.959} C_VEL
LIN {X 0,Y 544.685,Z 400.872,A -85,B 0,C 180,E1 -3694.069,E2 -3694.069} C_VEL
LIN {X 0,Y 544.654,Z 396.921,A -85,B 0,C 180,E1 -3695.182,E2 -3695.182} C_VEL
LIN {X 0,Y 544.726,Z 391.638,A -85,B 0,C 180,E1 -3696.333,E2 -3696.333} C_VEL
LIN {X 0,Y 544.84,Z 385.443,A -85,B 0,C 180,E1 -3697.411,E2 -3697.411} C_VEL
LIN {X 0,Y 545.005,Z 377.494,A -85,B 0,C 180,E1 -3698.528,E2 -3698.528} C_VEL
LIN {X 0,Y 545.139,Z 369.353,A -85,B 0,C 180,E1 -3699.461,E2 -3699.461} C_VEL
LIN {X 0,Y 545.331,Z 359.345,A -85,B 0,C 180,E1 -3700.394,E2 -3700.394} C_VEL
LIN {X 0,Y 545.519,Z 349.524,A -85,B 0,C 180,E1 -3701.142,E2 -3701.142} C_VEL
LIN {X 0,Y 545.686,Z 338.717,A -85,B 0,C 180,E1 -3701.809,E2 -3701.809} C_VEL
LIN {X 0,Y 545.918,Z 326.155,A -85,B 0,C 180,E1 -3702.405,E2 -3702.405} C_VEL
LIN {X 0,Y 546.103,Z 313.824,A -85,B 0,C 180,E1 -3702.826,E2 -3702.826} C_VEL
LIN {X 0,Y 545.934,Z 308.946,A -85,B 0,C 180,E1 -3702.96,E2 -3702.96} C_VEL
LIN {X 0,Y 544.634,Z 301.524,A -85,B 0,C 180,E1 -3703.146,E2 -3703.146} C_VEL
LIN {X 0,Y 544.682,Z 297.257,A -85,B 0,C 180,E1 -3704.955,E2 -3704.955} C_VEL
LIN {X 0,Y 544.738,Z 290.071,A -85,B 0,C 180,E1 -3708.037,E2 -3708.037} C_VEL
LIN {X 0,Y 544.823,Z 284.682,A -85,B 0,C 180,E1 -3710.382,E2 -3710.382} C_VEL
LIN {X 0,Y 544.87,Z 279.292,A -85,B 0,C 180,E1 -3712.765,E2 -3712.765} C_VEL
LIN {X 0,Y 544.94,Z 273.279,A -85,B 0,C 180,E1 -3715.472,E2 -3715.472} C_VEL
LIN {X 0,Y 544.983,Z 268.513,A -85,B 0,C 180,E1 -3717.661,E2 -3717.661} C_VEL
LIN {X 0,Y 545.086,Z 263.003,A -85,B 0,C 180,E1 -3720.245,E2 -3720.245} C_VEL
LIN {X 0,Y 545.197,Z 257.154,A -85,B 0,C 180,E1 -3723.079,E2 -3723.079} C_VEL
LIN {X 0,Y 545.279,Z 252.115,A -85,B 0,C 180,E1 -3725.706,E2 -3725.706} C_VEL
LIN {X 0,Y 545.448,Z 247.601,A -85,B 0,C 180,E1 -3728.204,E2 -3728.204} C_VEL
LIN {X 0,Y 545.585,Z 242.783,A -85,B 0,C 180,E1 -3731.068,E2 -3731.068} C_VEL
LIN {X 0,Y 545.289,Z 239.692,A -85,B 0,C 180,E1 -3733.085,E2 -3733.085} C_VEL
LIN {X 0,Y 545.031,Z 238.175,A -85,B 0,C 180,E1 -3734.131,E2 -3734.131} C_VEL
LIN {X 0,Y 545.023,Z 238.098,A -85,B 0,C 180,E1 -3736.885,E2 -3736.885} C_VEL
LIN {X 0,Y 545.055,Z 238.088,A -85,B 0,C 180,E1 -3739.854,E2 -3739.854} C_VEL
LIN {X 0,Y 545.068,Z 238.089,A -85,B 0,C 180,E1 -3743.073,E2 -3743.073} C_VEL
LIN {X 0,Y 545.049,Z 238.09,A -85,B 0,C 180,E1 -3746.324,E2 -3746.324} C_VEL
LIN {X 0,Y 545.057,Z 238.089,A -85,B 0,C 180,E1 -3748.949,E2 -3748.949} C_VEL
LIN {X 0,Y 545.041,Z 238.087,A -85,B 0,C 180,E1 -3751.501,E2 -3751.501} C_VEL
LIN {X 0,Y 545.038,Z 238.096,A -85,B 0,C 180,E1 -3754.502,E2 -3754.502} C_VEL
LIN {X 0,Y 545.028,Z 238.089,A -85,B 0,C 180,E1 -3757.239,E2 -3757.239} C_VEL
LIN {X 0,Y 545.103,Z 238.087,A -85,B 0,C 180,E1 -3760.411,E2 -3760.411} C_VEL
LIN {X 0,Y 545.018,Z 238.091,A -85,B 0,C 180,E1 -3763.516,E2 -3763.516} C_VEL
LIN {X 0,Y 545.079,Z 238.087,A -85,B 0,C 180,E1 -3765.816,E2 -3765.816} C_VEL
LIN {X 0,Y 545.113,Z 238.078,A -85,B 0,C 180,E1 -3768.846,E2 -3768.846} C_VEL
LIN {X 0,Y 545.064,Z 238.092,A -85,B 0,C 180,E1 -3771.842,E2 -3771.842} C_VEL
LIN {X 0,Y 545.163,Z 238.072,A -85,B 0,C 180,E1 -3774.819,E2 -3774.819} C_VEL
LIN {X 0,Y 545.178,Z 238.079,A -85,B 0,C 180,E1 -3777.779,E2 -3777.779} C_VEL
LIN {X 0,Y 545.177,Z 238.075,A -85,B 0,C 180,E1 -3779.996,E2 -3779.996} C_VEL
LIN {X 0,Y 545.149,Z 238.075,A -85,B 0,C 180,E1 -3782.951,E2 -3782.951} C_VEL
LIN {X 0,Y 545.12,Z 238.081,A -85,B 0,C 180,E1 -3785.915,E2 -3785.915} C_VEL
LIN {X 0,Y 545.076,Z 238.084,A -85,B 0,C 180,E1 -3788.149,E2 -3788.149} C_VEL
LIN {X 0,Y 545.119,Z 238.084,A -85,B 0,C 180,E1 -3791.531,E2 -3791.531} C_VEL
LIN {X 0,Y 545.056,Z 238.09,A -85,B 0,C 180,E1 -3794.939,E2 -3794.939} C_VEL
LIN {X 0,Y 545.038,Z 238.088,A -85,B 0,C 180,E1 -3798.022,E2 -3798.022} C_VEL
LIN {X 0,Y 545.065,Z 238.085,A -85,B 0,C 180,E1 -3800.367,E2 -3800.367} C_VEL
LIN {X 0,Y 545.05,Z 238.088,A -85,B 0,C 180,E1 -3803.555,E2 -3803.555} C_VEL
LIN {X 0,Y 545.046,Z 238.086,A -85,B 0,C 180,E1 -3805.996,E2 -3805.996} C_VEL
LIN {X 0,Y 545.055,Z 238.093,A -85,B 0,C 180,E1 -3808.743,E2 -3808.743} C_VEL
LIN {X 0,Y 545.02,Z 238.09,A -85,B 0,C 180,E1 -3811.674,E2 -3811.674} C_VEL
LIN {X 0,Y 545.042,Z 238.095,A -85,B 0,C 180,E1 -3814.558,E2 -3814.558} C_VEL
LIN {X 0,Y 545.027,Z 238.092,A -85,B 0,C 180,E1 -3816.968,E2 -3816.968} C_VEL
LIN {X 0,Y 544.314,Z 238.18,A -85,B 0,C 180,E1 -3817.584,E2 -3817.584} C_VEL
LIN {X 0,Y 541.443,Z 238.544,A -85,B 0,C 180,E1 -3818.585,E2 -3818.585} C_VEL
LIN {X 0,Y 539.059,Z 238.836,A -85,B 0,C 180,E1 -3819.391,E2 -3819.391} C_VEL
LIN {X 0,Y 538.058,Z 238.96,A -85,B 0,C 180,E1 -3820.013,E2 -3820.013} C_VEL
LIN {X 0,Y 537.986,Z 238.966,A -85,B 0,C 180,E1 -3820.224,E2 -3820.224} C_VEL
LIN {X 0,Y 537.988,Z 238.967,A -85,B 0,C 180,E1 -3822.984,E2 -3822.984} C_VEL
LIN {X 0,Y 537.978,Z 238.97,A -85,B 0,C 180,E1 -3825.921,E2 -3825.921} C_VEL
LIN {X 0,Y 538.026,Z 238.961,A -85,B 0,C 180,E1 -3829.245,E2 -3829.245} C_VEL
LIN {X 0,Y 537.94,Z 238.981,A -85,B 0,C 180,E1 -3832.119,E2 -3832.119} C_VEL
LIN {X 0,Y 537.965,Z 238.969,A -85,B 0,C 180,E1 -3834.914,E2 -3834.914} C_VEL
LIN {X 0,Y 537.975,Z 238.971,A -85,B 0,C 180,E1 -3837.615,E2 -3837.615} C_VEL
LIN {X 0,Y 537.986,Z 238.97,A -85,B 0,C 180,E1 -3840.238,E2 -3840.238} C_VEL
LIN {X 0,Y 538.01,Z 238.963,A -85,B 0,C 180,E1 -3842.794,E2 -3842.794} C_VEL
LIN {X 0,Y 538.01,Z 238.966,A -85,B 0,C 180,E1 -3845.291,E2 -3845.291} C_VEL
LIN {X 0,Y 537.983,Z 238.97,A -85,B 0,C 180,E1 -3848.03,E2 -3848.03} C_VEL
LIN {X 0,Y 537.979,Z 238.968,A -85,B 0,C 180,E1 -3850.938,E2 -3850.938} C_VEL
LIN {X 0,Y 537.995,Z 238.973,A -85,B 0,C 180,E1 -3853.298,E2 -3853.298} C_VEL
LIN {X 0,Y 538,Z 238.972,A -85,B 0,C 180,E1 -3855.629,E2 -3855.629} C_VEL
LIN {X 0,Y 538.031,Z 238.963,A -85,B 0,C 180,E1 -3858.701,E2 -3858.701} C_VEL
LIN {X 0,Y 538.029,Z 238.965,A -85,B 0,C 180,E1 -3861.739,E2 -3861.739} C_VEL
LIN {X 0,Y 538.067,Z 238.958,A -85,B 0,C 180,E1 -3864.002,E2 -3864.002} C_VEL
LIN {X 0,Y 538.084,Z 238.962,A -85,B 0,C 180,E1 -3867.005,E2 -3867.005} C_VEL
LIN {X 0,Y 538.1,Z 238.954,A -85,B 0,C 180,E1 -3870,E2 -3870} C_VEL
LIN {X 0,Y 538.084,Z 238.962,A -85,B 0,C 180,E1 -3872.995,E2 -3872.995} C_VEL
LIN {X 0,Y 538.067,Z 238.958,A -85,B 0,C 180,E1 -3875.998,E2 -3875.998} C_VEL
LIN {X 0,Y 538.029,Z 238.965,A -85,B 0,C 180,E1 -3878.261,E2 -3878.261} C_VEL
LIN {X 0,Y 538.031,Z 238.962,A -85,B 0,C 180,E1 -3881.608,E2 -3881.608} C_VEL
LIN {X 0,Y 538.016,Z 238.968,A -85,B 0,C 180,E1 -3884.87,E2 -3884.87} C_VEL
LIN {X 0,Y 538.026,Z 238.963,A -85,B 0,C 180,E1 -3887.554,E2 -3887.554} C_VEL
LIN {X 0,Y 537.98,Z 238.972,A -85,B 0,C 180,E1 -3890.653,E2 -3890.653} C_VEL
LIN {X 0,Y 538.013,Z 238.966,A -85,B 0,C 180,E1 -3893.887,E2 -3893.887} C_VEL
LIN {X 0,Y 537.996,Z 238.972,A -85,B 0,C 180,E1 -3896.369,E2 -3896.369} C_VEL
LIN {X 0,Y 537.995,Z 238.965,A -85,B 0,C 180,E1 -3898.942,E2 -3898.942} C_VEL
LIN {X 0,Y 537.973,Z 238.974,A -85,B 0,C 180,E1 -3901.895,E2 -3901.895} C_VEL
LIN {X 0,Y 537.978,Z 238.968,A -85,B 0,C 180,E1 -3904.625,E2 -3904.625} C_VEL
LIN {X 0,Y 537.953,Z 238.971,A -85,B 0,C 180,E1 -3907.174,E2 -3907.174} C_VEL
LIN {X 0,Y 538.003,Z 238.973,A -85,B 0,C 180,E1 -3909.798,E2 -3909.798} C_VEL
LIN {X 0,Y 537.972,Z 238.968,A -85,B 0,C 180,E1 -3912.79,E2 -3912.79} C_VEL
LIN {X 0,Y 537.982,Z 238.971,A -85,B 0,C 180,E1 -3915.93,E2 -3915.93} C_VEL
LIN {X 0,Y 538.032,Z 238.965,A -85,B 0,C 180,E1 -3919.254,E2 -3919.254} C_VEL
LIN {X 0,Y 537.95,Z 238.971,A -85,B 0,C 180,E1 -3922.127,E2 -3922.127} C_VEL
LIN {X 0,Y 537.98,Z 238.97,A -85,B 0,C 180,E1 -3924.922,E2 -3924.922} C_VEL
LIN {X 0,Y 537.98,Z 238.971,A -85,B 0,C 180,E1 -3927.622,E2 -3927.622} C_VEL
LIN {X 0,Y 537.982,Z 238.966,A -85,B 0,C 180,E1 -3930.244,E2 -3930.244} C_VEL
LIN {X 0,Y 538.034,Z 238.964,A -85,B 0,C 180,E1 -3932.801,E2 -3932.801} C_VEL
LIN {X 0,Y 537.992,Z 238.971,A -85,B 0,C 180,E1 -3935.296,E2 -3935.296} C_VEL
LIN {X 0,Y 537.987,Z 238.966,A -85,B 0,C 180,E1 -3938.047,E2 -3938.047} C_VEL
LIN {X 0,Y 538.054,Z 238.958,A -85,B 0,C 180,E1 -3940.153,E2 -3940.153} C_VEL
LIN {X 0,Y 537.987,Z 238.968,A -85,B 0,C 180,E1 -3943.303,E2 -3943.303} C_VEL
LIN {X 0,Y 538.019,Z 238.962,A -85,B 0,C 180,E1 -3945.635,E2 -3945.635} C_VEL
LIN {X 0,Y 538.061,Z 238.965,A -85,B 0,C 180,E1 -3948.706,E2 -3948.706} C_VEL
LIN {X 0,Y 538.041,Z 238.959,A -85,B 0,C 180,E1 -3951.744,E2 -3951.744} C_VEL
LIN {X 0,Y 538.134,Z 238.952,A -85,B 0,C 180,E1 -3954.759,E2 -3954.759} C_VEL
LIN {X 0,Y 538.146,Z 238.947,A -85,B 0,C 180,E1 -3957.759,E2 -3957.759} C_VEL
LIN {X 0,Y 538.169,Z 238.946,A -85,B 0,C 180,E1 -3960.753,E2 -3960.753} C_VEL
LIN {X 0,Y 538.111,Z 238.951,A -85,B 0,C 180,E1 -3962.999,E2 -3962.999} C_VEL
LIN {X 0,Y 538.078,Z 238.962,A -85,B 0,C 180,E1 -3966.002,E2 -3966.002} C_VEL
LIN {X 0,Y 538.042,Z 238.959,A -85,B 0,C 180,E1 -3969.022,E2 -3969.022} C_VEL
LIN {X 0,Y 538.057,Z 238.965,A -85,B 0,C 180,E1 -3972.067,E2 -3972.067} C_VEL
LIN {X 0,Y 538.037,Z 238.96,A -85,B 0,C 180,E1 -3975.148,E2 -3975.148} C_VEL
LIN {X 0,Y 538.002,Z 238.966,A -85,B 0,C 180,E1 -3978.275,E2 -3978.275} C_VEL
LIN {X 0,Y 538.007,Z 238.963,A -85,B 0,C 180,E1 -3980.656,E2 -3980.656} C_VEL
LIN {X 0,Y 538.007,Z 238.965,A -85,B 0,C 180,E1 -3983.075,E2 -3983.075} C_VEL
LIN {X 0,Y 537.997,Z 238.972,A -85,B 0,C 180,E1 -3985.664,E2 -3985.664} C_VEL
LIN {X 0,Y 537.978,Z 238.969,A -85,B 0,C 180,E1 -3988.056,E2 -3988.056} C_VEL
LIN {X 0,Y 538.007,Z 238.964,A -85,B 0,C 180,E1 -3990.631,E2 -3990.631} C_VEL
LIN {X 0,Y 538.025,Z 238.97,A -85,B 0,C 180,E1 -3993.281,E2 -3993.281} C_VEL
LIN {X 0,Y 537.974,Z 238.97,A -85,B 0,C 180,E1 -3996.009,E2 -3996.009} C_VEL
LIN {X 0,Y 538.011,Z 238.969,A -85,B 0,C 180,E1 -3998.833,E2 -3998.833} C_VEL
LIN {X 0,Y 537.989,Z 238.969,A -85,B 0,C 180,E1 -4001.875,E2 -4001.875} C_VEL
LIN {X 0,Y 537.999,Z 238.973,A -85,B 0,C 180,E1 -4004.866,E2 -4004.866} C_VEL
LIN {X 0,Y 538.137,Z 239.946,A -85,B 0,C 180,E1 -4006.199,E2 -4006.199} C_VEL
LIN {X 0,Y 538.544,Z 243.005,A -85,B 0,C 180,E1 -4008.276,E2 -4008.276} C_VEL
LIN {X 0,Y 538.525,Z 246.354,A -85,B 0,C 180,E1 -4010.354,E2 -4010.354} C_VEL
LIN {X 0,Y 538.354,Z 251.08,A -85,B 0,C 180,E1 -4013.094,E2 -4013.094} C_VEL
LIN {X 0,Y 538.194,Z 256.078,A -85,B 0,C 180,E1 -4015.84,E2 -4015.84} C_VEL
LIN {X 0,Y 538.073,Z 261.34,A -85,B 0,C 180,E1 -4018.503,E2 -4018.503} C_VEL
LIN {X 0,Y 537.991,Z 266.717,A -85,B 0,C 180,E1 -4021.096,E2 -4021.096} C_VEL
LIN {X 0,Y 537.918,Z 272.106,A -85,B 0,C 180,E1 -4023.627,E2 -4023.627} C_VEL
LIN {X 0,Y 537.83,Z 277.636,A -85,B 0,C 180,E1 -4026.168,E2 -4026.168} C_VEL
LIN {X 0,Y 537.791,Z 282.885,A -85,B 0,C 180,E1 -4028.537,E2 -4028.537} C_VEL
LIN {X 0,Y 537.709,Z 288.275,A -85,B 0,C 180,E1 -4030.928,E2 -4030.928} C_VEL
LIN {X 0,Y 537.644,Z 293.664,A -85,B 0,C 180,E1 -4033.287,E2 -4033.287} C_VEL
LIN {X 0,Y 537.638,Z 299.054,A -85,B 0,C 180,E1 -4035.619,E2 -4035.619} C_VEL
LIN {X 0,Y 537.579,Z 301.524,A -85,B 0,C 180,E1 -4036.678,E2 -4036.678} C_VEL
LIN {X 0,Y 539.202,Z 312.061,A -85,B 0,C 180,E1 -4036.959,E2 -4036.959} C_VEL
LIN {X 0,Y 539.032,Z 323.667,A -85,B 0,C 180,E1 -4037.338,E2 -4037.338} C_VEL
LIN {X 0,Y 538.816,Z 335.41,A -85,B 0,C 180,E1 -4037.859,E2 -4037.859} C_VEL
LIN {X 0,Y 538.623,Z 346.212,A -85,B 0,C 180,E1 -4038.486,E2 -4038.486} C_VEL
LIN {X 0,Y 538.372,Z 357.076,A -85,B 0,C 180,E1 -4039.279,E2 -4039.279} C_VEL
LIN {X 0,Y 538.196,Z 365.569,A -85,B 0,C 180,E1 -4040.036,E2 -4040.036} C_VEL
LIN {X 0,Y 538.014,Z 374.372,A -85,B 0,C 180,E1 -4040.982,E2 -4040.982} C_VEL
LIN {X 0,Y 537.832,Z 383.009,A -85,B 0,C 180,E1 -4042.114,E2 -4042.114} C_VEL
LIN {X 0,Y 537.702,Z 390.691,A -85,B 0,C 180,E1 -4043.398,E2 -4043.398} C_VEL
LIN {X 0,Y 537.674,Z 395.363,A -85,B 0,C 180,E1 -4044.374,E2 -4044.374} C_VEL
LIN {X 0,Y 537.558,Z 399.659,A -85,B 0,C 180,E1 -4045.501,E2 -4045.501} C_VEL
LIN {X 0,Y 537.592,Z 401.97,A -85,B 0,C 180,E1 -4046.252,E2 -4046.252} C_VEL
LIN {X 0,Y 537.553,Z 403.785,A -85,B 0,C 180,E1 -4047.002,E2 -4047.002} C_VEL
LIN {X 0,Y 537.452,Z 406.192,A -85,B 0,C 180,E1 -4048.501,E2 -4048.501} C_VEL
LIN {X 0,Y 537.442,Z 406.781,A -85,B 0,C 180,E1 -4049.251,E2 -4049.251} C_VEL
LIN {X 0,Y 537.442,Z 406.781,A -85,B 0,C 180,E1 -4050.749,E2 -4050.749} C_VEL
LIN {X 0,Y 537.452,Z 406.192,A -85,B 0,C 180,E1 -4051.499,E2 -4051.499} C_VEL
LIN {X 0,Y 537.553,Z 403.785,A -85,B 0,C 180,E1 -4052.998,E2 -4052.998} C_VEL
LIN {X 0,Y 537.605,Z 400.869,A -85,B 0,C 180,E1 -4054.123,E2 -4054.123} C_VEL
LIN {X 0,Y 537.588,Z 396.917,A -85,B 0,C 180,E1 -4055.251,E2 -4055.251} C_VEL
LIN {X 0,Y 537.641,Z 392.135,A -85,B 0,C 180,E1 -4056.317,E2 -4056.317} C_VEL
LIN {X 0,Y 537.758,Z 386.588,A -85,B 0,C 180,E1 -4057.321,E2 -4057.321} C_VEL
LIN {X 0,Y 537.885,Z 380.296,A -85,B 0,C 180,E1 -4058.263,E2 -4058.263} C_VEL
LIN {X 0,Y 538.026,Z 372.751,A -85,B 0,C 180,E1 -4059.208,E2 -4059.208} C_VEL
LIN {X 0,Y 538.227,Z 363.634,A -85,B 0,C 180,E1 -4060.153,E2 -4060.153} C_VEL
LIN {X 0,Y 538.478,Z 352.208,A -85,B 0,C 180,E1 -4061.099,E2 -4061.099} C_VEL
LIN {X 0,Y 538.663,Z 341.091,A -85,B 0,C 180,E1 -4061.826,E2 -4061.826} C_VEL
LIN {X 0,Y 538.894,Z 329.426,A -85,B 0,C 180,E1 -4062.426,E2 -4062.426} C_VEL
LIN {X 0,Y 539.165,Z 315.512,A -85,B 0,C 180,E1 -4062.946,E2 -4062.946} C_VEL
LIN {X 0,Y 538.977,Z 309.857,A -85,B 0,C 180,E1 -4063.106,E2 -4063.106} C_VEL
LIN {X 0,Y 537.579,Z 301.524,A -85,B 0,C 180,E1 -4063.322,E2 -4063.322} C_VEL
LIN {X 0,Y 537.621,Z 295.461,A -85,B 0,C 180,E1 -4065.933,E2 -4065.933} C_VEL
LIN {X 0,Y 537.663,Z 290.071,A -85,B 0,C 180,E1 -4068.283,E2 -4068.283} C_VEL
LIN {X 0,Y 537.761,Z 284.682,A -85,B 0,C 180,E1 -4070.662,E2 -4070.662} C_VEL
LIN {X 0,Y 537.797,Z 279.292,A -85,B 0,C 180,E1 -4073.081,E2 -4073.081} C_VEL
LIN {X 0,Y 537.889,Z 273.7,A -85,B 0,C 180,E1 -4075.635,E2 -4075.635} C_VEL
LIN {X 0,Y 537.963,Z 268.513,A -85,B 0,C 180,E1 -4078.054,E2 -4078.054} C_VEL
LIN {X 0,Y 538.036,Z 263.124,A -85,B 0,C 180,E1 -4080.625,E2 -4080.625} C_VEL
LIN {X 0,Y 538.173,Z 257.754,A -85,B 0,C 180,E1 -4083.301,E2 -4083.301} C_VEL
LIN {X 0,Y 538.278,Z 252.738,A -85,B 0,C 180,E1 -4085.982,E2 -4085.982} C_VEL
LIN {X 0,Y 538.495,Z 247.776,A -85,B 0,C 180,E1 -4088.788,E2 -4088.788} C_VEL
LIN {X 0,Y 538.593,Z 244.43,A -85,B 0,C 180,E1 -4090.812,E2 -4090.812} C_VEL
LIN {X 0,Y 538.336,Z 241.065,A -85,B 0,C 180,E1 -4093.02,E2 -4093.02} C_VEL
LIN {X 0,Y 538.083,Z 239.543,A -85,B 0,C 180,E1 -4094.078,E2 -4094.078} C_VEL
LIN {X 0,Y 537.999,Z 238.972,A -85,B 0,C 180,E1 -4095.134,E2 -4095.134} C_VEL
LIN {X 0,Y 537.988,Z 238.97,A -85,B 0,C 180,E1 -4098.22,E2 -4098.22} C_VEL
LIN {X 0,Y 538.011,Z 238.969,A -85,B 0,C 180,E1 -4101.167,E2 -4101.167} C_VEL
LIN {X 0,Y 537.973,Z 238.969,A -85,B 0,C 180,E1 -4104.09,E2 -4104.09} C_VEL
LIN {X 0,Y 538.036,Z 238.968,A -85,B 0,C 180,E1 -4106.725,E2 -4106.725} C_VEL
LIN {X 0,Y 538.007,Z 238.963,A -85,B 0,C 180,E1 -4109.558,E2 -4109.558} C_VEL
LIN {X 0,Y 537.978,Z 238.969,A -85,B 0,C 180,E1 -4111.944,E2 -4111.944} C_VEL
LIN {X 0,Y 538.019,Z 238.971,A -85,B 0,C 180,E1 -4114.461,E2 -4114.461} C_VEL
LIN {X 0,Y 538.007,Z 238.965,A -85,B 0,C 180,E1 -4116.925,E2 -4116.925} C_VEL
LIN {X 0,Y 538.044,Z 238.966,A -85,B 0,C 180,E1 -4120.143,E2 -4120.143} C_VEL
LIN {X 0,Y 537.99,Z 238.97,A -85,B 0,C 180,E1 -4122.511,E2 -4122.511} C_VEL
LIN {X 0,Y 538.049,Z 238.961,A -85,B 0,C 180,E1 -4125.627,E2 -4125.627} C_VEL
LIN {X 0,Y 538.073,Z 238.956,A -85,B 0,C 180,E1 -4128.698,E2 -4128.698} C_VEL
LIN {X 0,Y 538.035,Z 238.966,A -85,B 0,C 180,E1 -4131.735,E2 -4131.735} C_VEL
LIN {X 0,Y 538.121,Z 238.949,A -85,B 0,C 180,E1 -4134.751,E2 -4134.751} C_VEL
LIN {X 0,Y 538.151,Z 238.955,A -85,B 0,C 180,E1 -4137.75,E2 -4137.75} C_VEL
LIN {X 0,Y 538.146,Z 238.951,A -85,B 0,C 180,E1 -4139.996,E2 -4139.996} C_VEL
LIN {X 0,Y 538.116,Z 238.951,A -85,B 0,C 180,E1 -4142.99,E2 -4142.99} C_VEL
LIN {X 0,Y 538.076,Z 238.957,A -85,B 0,C 180,E1 -4145.993,E2 -4145.993} C_VEL
LIN {X 0,Y 538.041,Z 238.959,A -85,B 0,C 180,E1 -4148.256,E2 -4148.256} C_VEL
LIN {X 0,Y 538.069,Z 238.961,A -85,B 0,C 180,E1 -4151.594,E2 -4151.594} C_VEL
LIN {X 0,Y 538.021,Z 238.965,A -85,B 0,C 180,E1 -4154.846,E2 -4154.846} C_VEL
LIN {X 0,Y 538.012,Z 238.967,A -85,B 0,C 180,E1 -4157.527,E2 -4157.527} C_VEL
LIN {X 0,Y 538.01,Z 238.966,A -85,B 0,C 180,E1 -4160.647,E2 -4160.647} C_VEL
LIN {X 0,Y 537.972,Z 238.968,A -85,B 0,C 180,E1 -4163.884,E2 -4163.884} C_VEL
LIN {X 0,Y 538.009,Z 238.965,A -85,B 0,C 180,E1 -4166.362,E2 -4166.362} C_VEL
LIN {X 0,Y 537.996,Z 238.972,A -85,B 0,C 180,E1 -4168.929,E2 -4168.929} C_VEL
LIN {X 0,Y 537.973,Z 238.968,A -85,B 0,C 180,E1 -4171.882,E2 -4171.882} C_VEL
LIN {X 0,Y 537.992,Z 238.974,A -85,B 0,C 180,E1 -4174.616,E2 -4174.616} C_VEL
LIN {X 0,Y 537.965,Z 238.97,A -85,B 0,C 180,E1 -4177.166,E2 -4177.166} C_VEL
LIN {X 0,Y 537.986,Z 238.966,A -85,B 0,C 180,E1 -4180.224,E2 -4180.224} C_VEL
LIN {X 0,Y 537.346,Z 239.05,A -85,B 0,C 180,E1 -4180.849,E2 -4180.849} C_VEL
LIN {X 0,Y 534.496,Z 239.402,A -85,B 0,C 180,E1 -4181.864,E2 -4181.864} C_VEL
LIN {X 0,Y 532.064,Z 239.709,A -85,B 0,C 180,E1 -4182.681,E2 -4182.681} C_VEL
LIN {X 0,Y 531.009,Z 239.836,A -85,B 0,C 180,E1 -4183.312,E2 -4183.312} C_VEL
LIN {X 0,Y 530.918,Z 239.847,A -85,B 0,C 180,E1 -4183.526,E2 -4183.526} C_VEL
LIN {X 0,Y 530.915,Z 239.853,A -85,B 0,C 180,E1 -4186.501,E2 -4186.501} C_VEL
LIN {X 0,Y 530.956,Z 239.843,A -85,B 0,C 180,E1 -4189.566,E2 -4189.566} C_VEL
LIN {X 0,Y 530.914,Z 239.85,A -85,B 0,C 180,E1 -4192.573,E2 -4192.573} C_VEL
LIN {X 0,Y 530.947,Z 239.844,A -85,B 0,C 180,E1 -4195.308,E2 -4195.308} C_VEL
LIN {X 0,Y 530.927,Z 239.853,A -85,B 0,C 180,E1 -4198.03,E2 -4198.03} C_VEL
LIN {X 0,Y 530.946,Z 239.843,A -85,B 0,C 180,E1 -4200.867,E2 -4200.867} C_VEL
LIN {X 0,Y 530.954,Z 239.844,A -85,B 0,C 180,E1 -4203.254,E2 -4203.254} C_VEL
LIN {X 0,Y 530.964,Z 239.846,A -85,B 0,C 180,E1 -4205.947,E2 -4205.947} C_VEL
LIN {X 0,Y 530.944,Z 239.845,A -85,B 0,C 180,E1 -4209.06,E2 -4209.06} C_VEL
LIN {X 0,Y 530.984,Z 239.84,A -85,B 0,C 180,E1 -4212.334,E2 -4212.334} C_VEL
LIN {X 0,Y 530.984,Z 239.848,A -85,B 0,C 180,E1 -4215.435,E2 -4215.435} C_VEL
LIN {X 0,Y 530.985,Z 239.84,A -85,B 0,C 180,E1 -4218.549,E2 -4218.549} C_VEL
LIN {X 0,Y 530.998,Z 239.842,A -85,B 0,C 180,E1 -4221.629,E2 -4221.629} C_VEL
LIN {X 0,Y 531.025,Z 239.835,A -85,B 0,C 180,E1 -4223.922,E2 -4223.922} C_VEL
LIN {X 0,Y 531.049,Z 239.838,A -85,B 0,C 180,E1 -4226.966,E2 -4226.966} C_VEL
LIN {X 0,Y 531.071,Z 239.83,A -85,B 0,C 180,E1 -4230,E2 -4230} C_VEL
LIN {X 0,Y 531.049,Z 239.838,A -85,B 0,C 180,E1 -4233.034,E2 -4233.034} C_VEL
LIN {X 0,Y 531.025,Z 239.835,A -85,B 0,C 180,E1 -4236.078,E2 -4236.078} C_VEL
LIN {X 0,Y 530.998,Z 239.842,A -85,B 0,C 180,E1 -4238.371,E2 -4238.371} C_VEL
LIN {X 0,Y 530.994,Z 239.838,A -85,B 0,C 180,E1 -4241.68,E2 -4241.68} C_VEL
LIN {X 0,Y 530.981,Z 239.844,A -85,B 0,C 180,E1 -4244.965,E2 -4244.965} C_VEL
LIN {X 0,Y 530.963,Z 239.843,A -85,B 0,C 180,E1 -4247.724,E2 -4247.724} C_VEL
LIN {X 0,Y 530.944,Z 239.845,A -85,B 0,C 180,E1 -4250.94,E2 -4250.94} C_VEL
LIN {X 0,Y 530.964,Z 239.846,A -85,B 0,C 180,E1 -4254.053,E2 -4254.053} C_VEL
LIN {X 0,Y 530.954,Z 239.844,A -85,B 0,C 180,E1 -4256.746,E2 -4256.746} C_VEL
LIN {X 0,Y 530.941,Z 239.844,A -85,B 0,C 180,E1 -4259.325,E2 -4259.325} C_VEL
LIN {X 0,Y 530.925,Z 239.854,A -85,B 0,C 180,E1 -4262.107,E2 -4262.107} C_VEL
LIN {X 0,Y 530.934,Z 239.845,A -85,B 0,C 180,E1 -4264.858,E2 -4264.858} C_VEL
LIN {X 0,Y 530.912,Z 239.851,A -85,B 0,C 180,E1 -4267.511,E2 -4267.511} C_VEL
LIN {X 0,Y 530.956,Z 239.843,A -85,B 0,C 180,E1 -4270.434,E2 -4270.434} C_VEL
LIN {X 0,Y 530.915,Z 239.853,A -85,B 0,C 180,E1 -4273.499,E2 -4273.499} C_VEL
LIN {X 0,Y 530.92,Z 239.846,A -85,B 0,C 180,E1 -4276.51,E2 -4276.51} C_VEL
LIN {X 0,Y 530.955,Z 239.85,A -85,B 0,C 180,E1 -4279.573,E2 -4279.573} C_VEL
LIN {X 0,Y 530.927,Z 239.846,A -85,B 0,C 180,E1 -4282.582,E2 -4282.582} C_VEL
LIN {X 0,Y 530.962,Z 239.85,A -85,B 0,C 180,E1 -4285.316,E2 -4285.316} C_VEL
LIN {X 0,Y 530.929,Z 239.846,A -85,B 0,C 180,E1 -4288.037,E2 -4288.037} C_VEL
LIN {X 0,Y 530.955,Z 239.846,A -85,B 0,C 180,E1 -4290.879,E2 -4290.879} C_VEL
LIN {X 0,Y 530.973,Z 239.846,A -85,B 0,C 180,E1 -4293.261,E2 -4293.261} C_VEL
LIN {X 0,Y 530.929,Z 239.845,A -85,B 0,C 180,E1 -4295.972,E2 -4295.972} C_VEL
LIN {X 0,Y 530.971,Z 239.847,A -85,B 0,C 180,E1 -4299.067,E2 -4299.067} C_VEL
LIN {X 0,Y 530.951,Z 239.844,A -85,B 0,C 180,E1 -4301.483,E2 -4301.483} C_VEL
LIN {X 0,Y 530.97,Z 239.847,A -85,B 0,C 180,E1 -4304.655,E2 -4304.655} C_VEL
LIN {X 0,Y 531.008,Z 239.835,A -85,B 0,C 180,E1 -4307.78,E2 -4307.78} C_VEL
LIN {X 0,Y 530.96,Z 239.843,A -85,B 0,C 180,E1 -4310.097,E2 -4310.097} C_VEL
LIN {X 0,Y 531.057,Z 239.832,A -85,B 0,C 180,E1 -4312.993,E2 -4312.993} C_VEL
LIN {X 0,Y 531.092,Z 239.831,A -85,B 0,C 180,E1 -4314.69,E2 -4314.69} C_VEL
LIN {X 0,Y 531.119,Z 239.823,A -85,B 0,C 180,E1 -4317.729,E2 -4317.729} C_VEL
LIN {X 0,Y 531.14,Z 239.821,A -85,B 0,C 180,E1 -4320.763,E2 -4320.763} C_VEL
LIN {X 0,Y 531.052,Z 239.83,A -85,B 0,C 180,E1 -4323.039,E2 -4323.039} C_VEL
LIN {X 0,Y 531.038,Z 239.84,A -85,B 0,C 180,E1 -4326.082,E2 -4326.082} C_VEL
LIN {X 0,Y 531.004,Z 239.836,A -85,B 0,C 180,E1 -4329.143,E2 -4329.143} C_VEL
LIN {X 0,Y 531.047,Z 239.835,A -85,B 0,C 180,E1 -4331.674,E2 -4331.674} C_VEL
LIN {X 0,Y 531.022,Z 239.833,A -85,B 0,C 180,E1 -4334.956,E2 -4334.956} C_VEL
LIN {X 0,Y 530.964,Z 239.841,A -85,B 0,C 180,E1 -4338.526,E2 -4338.526} C_VEL
LIN {X 0,Y 530.979,Z 239.839,A -85,B 0,C 180,E1 -4340.942,E2 -4340.942} C_VEL
LIN {X 0,Y 530.956,Z 239.845,A -85,B 0,C 180,E1 -4344.034,E2 -4344.034} C_VEL
LIN {X 0,Y 530.95,Z 239.843,A -85,B 0,C 180,E1 -4346.75,E2 -4346.75} C_VEL
LIN {X 0,Y 530.965,Z 239.848,A -85,B 0,C 180,E1 -4349.327,E2 -4349.327} C_VEL
LIN {X 0,Y 530.961,Z 239.842,A -85,B 0,C 180,E1 -4352.101,E2 -4352.101} C_VEL
LIN {X 0,Y 530.961,Z 239.846,A -85,B 0,C 180,E1 -4354.851,E2 -4354.851} C_VEL
LIN {X 0,Y 530.967,Z 239.847,A -85,B 0,C 180,E1 -4357.51,E2 -4357.51} C_VEL
LIN {X 0,Y 530.955,Z 239.846,A -85,B 0,C 180,E1 -4360.438,E2 -4360.438} C_VEL
LIN {X 0,Y 530.932,Z 239.852,A -85,B 0,C 180,E1 -4363.501,E2 -4363.501} C_VEL
LIN {X 0,Y 530.969,Z 239.848,A -85,B 0,C 180,E1 -4364.552,E2 -4364.552} C_VEL
LIN {X 0,Y 531.038,Z 240.416,A -85,B 0,C 180,E1 -4365.618,E2 -4365.618} C_VEL
LIN {X 0,Y 531.462,Z 243.517,A -85,B 0,C 180,E1 -4367.78,E2 -4367.78} C_VEL
LIN {X 0,Y 531.529,Z 247.106,A -85,B 0,C 180,E1 -4370.078,E2 -4370.078} C_VEL
LIN {X 0,Y 531.386,Z 251.227,A -85,B 0,C 180,E1 -4372.528,E2 -4372.528} C_VEL
LIN {X 0,Y 531.192,Z 256.221,A -85,B 0,C 180,E1 -4375.326,E2 -4375.326} C_VEL
LIN {X 0,Y 531.094,Z 261.418,A -85,B 0,C 180,E1 -4378.041,E2 -4378.041} C_VEL
LIN {X 0,Y 530.972,Z 267.136,A -85,B 0,C 180,E1 -4380.88,E2 -4380.88} C_VEL
LIN {X 0,Y 530.853,Z 273.903,A -85,B 0,C 180,E1 -4384.095,E2 -4384.095} C_VEL
LIN {X 0,Y 530.74,Z 279.292,A -85,B 0,C 180,E1 -4386.594,E2 -4386.594} C_VEL
LIN {X 0,Y 530.712,Z 284.682,A -85,B 0,C 180,E1 -4389.051,E2 -4389.051} C_VEL
LIN {X 0,Y 530.59,Z 290.071,A -85,B 0,C 180,E1 -4391.465,E2 -4391.465} C_VEL
LIN {X 0,Y 530.535,Z 295.461,A -85,B 0,C 180,E1 -4393.848,E2 -4393.848} C_VEL
LIN {X 0,Y 530.497,Z 301.299,A -85,B 0,C 180,E1 -4396.4,E2 -4396.4} C_VEL
LIN {X 0,Y 530.478,Z 301.524,A -85,B 0,C 180,E1 -4396.497,E2 -4396.497} C_VEL
LIN {X 0,Y 532.302,Z 312.919,A -85,B 0,C 180,E1 -4396.811,E2 -4396.811} C_VEL
LIN {X 0,Y 532.097,Z 324.943,A -85,B 0,C 180,E1 -4397.219,E2 -4397.219} C_VEL
LIN {X 0,Y 531.802,Z 337.202,A -85,B 0,C 180,E1 -4397.793,E2 -4397.793} C_VEL
LIN {X 0,Y 531.596,Z 348.088,A -85,B 0,C 180,E1 -4398.46,E2 -4398.46} C_VEL
LIN {X 0,Y 531.352,Z 358.201,A -85,B 0,C 180,E1 -4399.233,E2 -4399.233} C_VEL
LIN {X 0,Y 531.11,Z 367.476,A -85,B 0,C 180,E1 -4400.095,E2 -4400.095} C_VEL
LIN {X 0,Y 530.931,Z 375.988,A -85,B 0,C 180,E1 -4401.052,E2 -4401.052} C_VEL
LIN {X 0,Y 530.762,Z 384.251,A -85,B 0,C 180,E1 -4402.2,E2 -4402.2} C_VEL
LIN {X 0,Y 530.6,Z 391.256,A -85,B 0,C 180,E1 -4403.423,E2 -4403.423} C_VEL
LIN {X 0,Y 530.524,Z 396.912,A -85,B 0,C 180,E1 -4404.679,E2 -4404.679} C_VEL
LIN {X 0,Y 530.524,Z 400.865,A -85,B 0,C 180,E1 -4405.822,E2 -4405.822} C_VEL
LIN {X 0,Y 530.459,Z 403.782,A -85,B 0,C 180,E1 -4406.962,E2 -4406.962} C_VEL
LIN {X 0,Y 530.362,Z 406.193,A -85,B 0,C 180,E1 -4408.481,E2 -4408.481} C_VEL
LIN {X 0,Y 530.344,Z 406.781,A -85,B 0,C 180,E1 -4409.241,E2 -4409.241} C_VEL
LIN {X 0,Y 530.344,Z 406.781,A -85,B 0,C 180,E1 -4410.759,E2 -4410.759} C_VEL
LIN {X 0,Y 530.362,Z 406.193,A -85,B 0,C 180,E1 -4411.519,E2 -4411.519} C_VEL
LIN {X 0,Y 530.459,Z 403.782,A -85,B 0,C 180,E1 -4413.038,E2 -4413.038} C_VEL
LIN {X 0,Y 530.524,Z 400.865,A -85,B 0,C 180,E1 -4414.178,E2 -4414.178} C_VEL
LIN {X 0,Y 530.524,Z 396.912,A -85,B 0,C 180,E1 -4415.321,E2 -4415.321} C_VEL
LIN {X 0,Y 530.597,Z 391.27,A -85,B 0,C 180,E1 -4416.574,E2 -4416.574} C_VEL
LIN {X 0,Y 530.762,Z 384.251,A -85,B 0,C 180,E1 -4417.8,E2 -4417.8} C_VEL
LIN {X 0,Y 530.931,Z 375.988,A -85,B 0,C 180,E1 -4418.948,E2 -4418.948} C_VEL
LIN {X 0,Y 531.109,Z 367.476,A -85,B 0,C 180,E1 -4419.905,E2 -4419.905} C_VEL
LIN {X 0,Y 531.348,Z 358.201,A -85,B 0,C 180,E1 -4420.768,E2 -4420.768} C_VEL
LIN {X 0,Y 531.604,Z 348.078,A -85,B 0,C 180,E1 -4421.54,E2 -4421.54} C_VEL
LIN {X 0,Y 531.8,Z 337.202,A -85,B 0,C 180,E1 -4422.207,E2 -4422.207} C_VEL
LIN {X 0,Y 532.087,Z 324.943,A -85,B 0,C 180,E1 -4422.782,E2 -4422.782} C_VEL
LIN {X 0,Y 532.294,Z 312.919,A -85,B 0,C 180,E1 -4423.189,E2 -4423.189} C_VEL
LIN {X 0,Y 530.478,Z 301.524,A -85,B 0,C 180,E1 -4423.503,E2 -4423.503} C_VEL
LIN {X 0,Y 530.528,Z 297.257,A -85,B 0,C 180,E1 -4425.363,E2 -4425.363} C_VEL
LIN {X 0,Y 530.599,Z 291.868,A -85,B 0,C 180,E1 -4427.736,E2 -4427.736} C_VEL
LIN {X 0,Y 530.69,Z 286.478,A -85,B 0,C 180,E1 -4430.14,E2 -4430.14} C_VEL
LIN {X 0,Y 530.738,Z 281.089,A -85,B 0,C 180,E1 -4432.582,E2 -4432.582} C_VEL
LIN {X 0,Y 530.793,Z 275.699,A -85,B 0,C 180,E1 -4435.068,E2 -4435.068} C_VEL
LIN {X 0,Y 530.901,Z 270.31,A -85,B 0,C 180,E1 -4437.601,E2 -4437.601} C_VEL
LIN {X 0,Y 530.976,Z 264.931,A -85,B 0,C 180,E1 -4440.196,E2 -4440.196} C_VEL
LIN {X 0,Y 531.112,Z 259.664,A -85,B 0,C 180,E1 -4442.856,E2 -4442.856} C_VEL
LIN {X 0,Y 531.247,Z 254.555,A -85,B 0,C 180,E1 -4445.597,E2 -4445.597} C_VEL
LIN {X 0,Y 531.481,Z 249.559,A -85,B 0,C 180,E1 -4448.425,E2 -4448.425} C_VEL
LIN {X 0,Y 531.574,Z 244.772,A -85,B 0,C 180,E1 -4451.379,E2 -4451.379} C_VEL
LIN {X 0,Y 531.235,Z 241.693,A -85,B 0,C 180,E1 -4453.466,E2 -4453.466} C_VEL
LIN {X 0,Y 530.989,Z 240.179,A -85,B 0,C 180,E1 -4454.546,E2 -4454.546} C_VEL
LIN {X 0,Y 530.932,Z 239.851,A -85,B 0,C 180,E1 -4456.499,E2 -4456.499} C_VEL
LIN {X 0,Y 530.946,Z 239.847,A -85,B 0,C 180,E1 -4459.561,E2 -4459.561} C_VEL
LIN {X 0,Y 530.969,Z 239.848,A -85,B 0,C 180,E1 -4462.576,E2 -4462.576} C_VEL
LIN {X 0,Y 530.972,Z 239.841,A -85,B 0,C 180,E1 -4465.306,E2 -4465.306} C_VEL
LIN {X 0,Y 530.961,Z 239.842,A -85,B 0,C 180,E1 -4468.028,E2 -4468.028} C_VEL
LIN {X 0,Y 530.967,Z 239.845,A -85,B 0,C 180,E1 -4470.877,E2 -4470.877} C_VEL
LIN {X 0,Y 530.95,Z 239.843,A -85,B 0,C 180,E1 -4473.25,E2 -4473.25} C_VEL
LIN {X 0,Y 530.956,Z 239.845,A -85,B 0,C 180,E1 -4475.966,E2 -4475.966} C_VEL
LIN {X 0,Y 530.979,Z 239.839,A -85,B 0,C 180,E1 -4479.058,E2 -4479.058} C_VEL
LIN {X 0,Y 530.964,Z 239.841,A -85,B 0,C 180,E1 -4481.474,E2 -4481.474} C_VEL
LIN {X 0,Y 531.022,Z 239.833,A -85,B 0,C 180,E1 -4485.044,E2 -4485.044} C_VEL
LIN {X 0,Y 531.032,Z 239.834,A -85,B 0,C 180,E1 -4488.546,E2 -4488.546} C_VEL
LIN {X 0,Y 530.986,Z 239.842,A -85,B 0,C 180,E1 -4491.624,E2 -4491.624} C_VEL
LIN {X 0,Y 531.082,Z 239.826,A -85,B 0,C 180,E1 -4494.681,E2 -4494.681} C_VEL
LIN {X 0,Y 531.123,Z 239.83,A -85,B 0,C 180,E1 -4497.721,E2 -4497.721} C_VEL
LIN {X 0,Y 531.115,Z 239.826,A -85,B 0,C 180,E1 -4499.996,E2 -4499.996} C_VEL
LIN {X 0,Y 531.084,Z 239.828,A -85,B 0,C 180,E1 -4503.03,E2 -4503.03} C_VEL
LIN {X 0,Y 531.036,Z 239.834,A -85,B 0,C 180,E1 -4506.073,E2 -4506.073} C_VEL
LIN {X 0,Y 530.994,Z 239.842,A -85,B 0,C 180,E1 -4509.134,E2 -4509.134} C_VEL
LIN {X 0,Y 531.032,Z 239.836,A -85,B 0,C 180,E1 -4511.666,E2 -4511.666} C_VEL
LIN {X 0,Y 530.997,Z 239.841,A -85,B 0,C 180,E1 -4514.946,E2 -4514.946} C_VEL
LIN {X 0,Y 530.956,Z 239.843,A -85,B 0,C 180,E1 -4517.719,E2 -4517.719} C_VEL
LIN {X 0,Y 530.999,Z 239.836,A -85,B 0,C 180,E1 -4520.122,E2 -4520.122} C_VEL
LIN {X 0,Y 530.917,Z 239.85,A -85,B 0,C 180,E1 -4522.568,E2 -4522.568} C_VEL
LIN {X 0,Y 530.958,Z 239.849,A -85,B 0,C 180,E1 -4525.053,E2 -4525.053} C_VEL
LIN {X 0,Y 530.983,Z 239.839,A -85,B 0,C 180,E1 -4527.59,E2 -4527.59} C_VEL
LIN {X 0,Y 530.938,Z 239.851,A -85,B 0,C 180,E1 -4530.64,E2 -4530.64} C_VEL
LIN {X 0,Y 530.951,Z 239.842,A -85,B 0,C 180,E1 -4533.768,E2 -4533.768} C_VEL
LIN {X 0,Y 530.927,Z 239.854,A -85,B 0,C 180,E1 -4536.553,E2 -4536.553} C_VEL
LIN {X 0,Y 530.937,Z 239.845,A -85,B 0,C 180,E1 -4539.85,E2 -4539.85} C_VEL
LIN {X 0,Y 530.937,Z 239.853,A -85,B 0,C 180,E1 -4542.452,E2 -4542.452} C_VEL
LIN {X 0,Y 530.918,Z 239.847,A -85,B 0,C 180,E1 -4543.526,E2 -4543.526} C_VEL
LIN {X 0,Y 530.242,Z 239.938,A -85,B 0,C 180,E1 -4544.159,E2 -4544.159} C_VEL
LIN {X 0,Y 527.394,Z 240.291,A -85,B 0,C 180,E1 -4545.188,E2 -4545.188} C_VEL
LIN {X 0,Y 524.992,Z 240.591,A -85,B 0,C 180,E1 -4546.016,E2 -4546.016} C_VEL
LIN {X 0,Y 523.958,Z 240.718,A -85,B 0,C 180,E1 -4546.656,E2 -4546.656} C_VEL
LIN {X 0,Y 523.872,Z 240.726,A -85,B 0,C 180,E1 -4546.872,E2 -4546.872} C_VEL
LIN {X 0,Y 523.926,Z 240.722,A -85,B 0,C 180,E1 -4549.919,E2 -4549.919} C_VEL
LIN {X 0,Y 523.856,Z 240.727,A -85,B 0,C 180,E1 -4552.864,E2 -4552.864} C_VEL
LIN {X 0,Y 523.889,Z 240.726,A -85,B 0,C 180,E1 -4555.707,E2 -4555.707} C_VEL
LIN {X 0,Y 523.877,Z 240.726,A -85,B 0,C 180,E1 -4558.454,E2 -4558.454} C_VEL
LIN {X 0,Y 523.891,Z 240.722,A -85,B 0,C 180,E1 -4561.123,E2 -4561.123} C_VEL
LIN {X 0,Y 523.928,Z 240.723,A -85,B 0,C 180,E1 -4563.976,E2 -4563.976} C_VEL
LIN {X 0,Y 523.909,Z 240.721,A -85,B 0,C 180,E1 -4566.27,E2 -4566.27} C_VEL
LIN {X 0,Y 523.895,Z 240.721,A -85,B 0,C 180,E1 -4568.765,E2 -4568.765} C_VEL
LIN {X 0,Y 523.894,Z 240.725,A -85,B 0,C 180,E1 -4571.219,E2 -4571.219} C_VEL
LIN {X 0,Y 523.896,Z 240.729,A -85,B 0,C 180,E1 -4573.638,E2 -4573.638} C_VEL
LIN {X 0,Y 523.888,Z 240.726,A -85,B 0,C 180,E1 -4576.027,E2 -4576.027} C_VEL
LIN {X 0,Y 523.945,Z 240.717,A -85,B 0,C 180,E1 -4578.393,E2 -4578.393} C_VEL
LIN {X 0,Y 523.945,Z 240.722,A -85,B 0,C 180,E1 -4581.515,E2 -4581.515} C_VEL
LIN {X 0,Y 523.986,Z 240.713,A -85,B 0,C 180,E1 -4583.84,E2 -4583.84} C_VEL
LIN {X 0,Y 524.015,Z 240.714,A -85,B 0,C 180,E1 -4586.925,E2 -4586.925} C_VEL
LIN {X 0,Y 524.042,Z 240.706,A -85,B 0,C 180,E1 -4590,E2 -4590} C_VEL
LIN {X 0,Y 524.015,Z 240.714,A -85,B 0,C 180,E1 -4593.075,E2 -4593.075} C_VEL
LIN {X 0,Y 523.986,Z 240.713,A -85,B 0,C 180,E1 -4596.16,E2 -4596.16} C_VEL
LIN {X 0,Y 523.945,Z 240.722,A -85,B 0,C 180,E1 -4598.485,E2 -4598.485} C_VEL
LIN {X 0,Y 523.955,Z 240.715,A -85,B 0,C 180,E1 -4601.753,E2 -4601.753} C_VEL
LIN {X 0,Y 523.94,Z 240.72,A -85,B 0,C 180,E1 -4605.06,E2 -4605.06} C_VEL
LIN {X 0,Y 523.905,Z 240.724,A -85,B 0,C 180,E1 -4607.971,E2 -4607.971} C_VEL
LIN {X 0,Y 523.909,Z 240.729,A -85,B 0,C 180,E1 -4610.412,E2 -4610.412} C_VEL
LIN {X 0,Y 523.901,Z 240.722,A -85,B 0,C 180,E1 -4612.894,E2 -4612.894} C_VEL
LIN {X 0,Y 523.922,Z 240.718,A -85,B 0,C 180,E1 -4615.42,E2 -4615.42} C_VEL
LIN {X 0,Y 523.91,Z 240.726,A -85,B 0,C 180,E1 -4618.002,E2 -4618.002} C_VEL
LIN {X 0,Y 523.91,Z 240.72,A -85,B 0,C 180,E1 -4620.863,E2 -4620.863} C_VEL
LIN {X 0,Y 523.905,Z 240.725,A -85,B 0,C 180,E1 -4623.739,E2 -4623.739} C_VEL
LIN {X 0,Y 523.866,Z 240.727,A -85,B 0,C 180,E1 -4626.408,E2 -4626.408} C_VEL
LIN {X 0,Y 523.907,Z 240.72,A -85,B 0,C 180,E1 -4629.085,E2 -4629.085} C_VEL
LIN {X 0,Y 523.907,Z 240.723,A -85,B 0,C 180,E1 -4632.122,E2 -4632.122} C_VEL
LIN {X 0,Y 523.907,Z 240.724,A -85,B 0,C 180,E1 -4635.313,E2 -4635.313} C_VEL
LIN {X 0,Y 523.927,Z 240.718,A -85,B 0,C 180,E1 -4638.692,E2 -4638.692} C_VEL
LIN {X 0,Y 523.873,Z 240.727,A -85,B 0,C 180,E1 -4641.903,E2 -4641.903} C_VEL
LIN {X 0,Y 523.899,Z 240.724,A -85,B 0,C 180,E1 -4644.914,E2 -4644.914} C_VEL
LIN {X 0,Y 523.897,Z 240.724,A -85,B 0,C 180,E1 -4647.685,E2 -4647.685} C_VEL
LIN {X 0,Y 523.92,Z 240.72,A -85,B 0,C 180,E1 -4650.681,E2 -4650.681} C_VEL
LIN {X 0,Y 523.921,Z 240.723,A -85,B 0,C 180,E1 -4652.872,E2 -4652.872} C_VEL
LIN {X 0,Y 523.91,Z 240.72,A -85,B 0,C 180,E1 -4655.807,E2 -4655.807} C_VEL
LIN {X 0,Y 523.918,Z 240.725,A -85,B 0,C 180,E1 -4658.772,E2 -4658.772} C_VEL
LIN {X 0,Y 523.914,Z 240.723,A -85,B 0,C 180,E1 -4661.225,E2 -4661.225} C_VEL
LIN {X 0,Y 523.903,Z 240.721,A -85,B 0,C 180,E1 -4663.643,E2 -4663.643} C_VEL
LIN {X 0,Y 523.896,Z 240.722,A -85,B 0,C 180,E1 -4666.032,E2 -4666.032} C_VEL
LIN {X 0,Y 523.995,Z 240.714,A -85,B 0,C 180,E1 -4668.399,E2 -4668.399} C_VEL
LIN {X 0,Y 523.968,Z 240.712,A -85,B 0,C 180,E1 -4671.52,E2 -4671.52} C_VEL
LIN {X 0,Y 524.002,Z 240.709,A -85,B 0,C 180,E1 -4673.845,E2 -4673.845} C_VEL
LIN {X 0,Y 524.026,Z 240.707,A -85,B 0,C 180,E1 -4676.929,E2 -4676.929} C_VEL
LIN {X 0,Y 523.985,Z 240.718,A -85,B 0,C 180,E1 -4678.467,E2 -4678.467} C_VEL
LIN {X 0,Y 524.11,Z 240.697,A -85,B 0,C 180,E1 -4680.773,E2 -4680.773} C_VEL
LIN {X 0,Y 523.995,Z 240.709,A -85,B 0,C 180,E1 -4683.08,E2 -4683.08} C_VEL
LIN {X 0,Y 523.999,Z 240.717,A -85,B 0,C 180,E1 -4686.164,E2 -4686.164} C_VEL
LIN {X 0,Y 523.975,Z 240.712,A -85,B 0,C 180,E1 -4689.266,E2 -4689.266} C_VEL
LIN {X 0,Y 523.996,Z 240.714,A -85,B 0,C 180,E1 -4691.74,E2 -4691.74} C_VEL
LIN {X 0,Y 523.986,Z 240.71,A -85,B 0,C 180,E1 -4695.053,E2 -4695.053} C_VEL
LIN {X 0,Y 523.914,Z 240.725,A -85,B 0,C 180,E1 -4697.974,E2 -4697.974} C_VEL
LIN {X 0,Y 523.946,Z 240.716,A -85,B 0,C 180,E1 -4700.415,E2 -4700.415} C_VEL
LIN {X 0,Y 523.908,Z 240.72,A -85,B 0,C 180,E1 -4702.897,E2 -4702.897} C_VEL
LIN {X 0,Y 523.902,Z 240.728,A -85,B 0,C 180,E1 -4705.425,E2 -4705.425} C_VEL
LIN {X 0,Y 523.903,Z 240.722,A -85,B 0,C 180,E1 -4708.006,E2 -4708.006} C_VEL
LIN {X 0,Y 523.913,Z 240.721,A -85,B 0,C 180,E1 -4710.851,E2 -4710.851} C_VEL
LIN {X 0,Y 523.931,Z 240.722,A -85,B 0,C 180,E1 -4713.731,E2 -4713.731} C_VEL
LIN {X 0,Y 523.892,Z 240.724,A -85,B 0,C 180,E1 -4716.401,E2 -4716.401} C_VEL
LIN {X 0,Y 523.916,Z 240.728,A -85,B 0,C 180,E1 -4719.088,E2 -4719.088} C_VEL
LIN {X 0,Y 523.901,Z 240.724,A -85,B 0,C 180,E1 -4722.127,E2 -4722.127} C_VEL
LIN {X 0,Y 523.922,Z 240.726,A -85,B 0,C 180,E1 -4724.689,E2 -4724.689} C_VEL
LIN {X 0,Y 524.202,Z 242.767,A -85,B 0,C 180,E1 -4726.387,E2 -4726.387} C_VEL
LIN {X 0,Y 524.587,Z 246.011,A -85,B 0,C 180,E1 -4728.614,E2 -4728.614} C_VEL
LIN {X 0,Y 524.478,Z 249.818,A -85,B 0,C 180,E1 -4731.008,E2 -4731.008} C_VEL
LIN {X 0,Y 524.295,Z 254.149,A -85,B 0,C 180,E1 -4733.543,E2 -4733.543} C_VEL
LIN {X 0,Y 524.117,Z 259.743,A -85,B 0,C 180,E1 -4736.649,E2 -4736.649} C_VEL
LIN {X 0,Y 523.996,Z 265.009,A -85,B 0,C 180,E1 -4739.359,E2 -4739.359} C_VEL
LIN {X 0,Y 523.857,Z 270.959,A -85,B 0,C 180,E1 -4742.309,E2 -4742.309} C_VEL
LIN {X 0,Y 523.748,Z 275.699,A -85,B 0,C 180,E1 -4744.571,E2 -4744.571} C_VEL
LIN {X 0,Y 523.686,Z 281.089,A -85,B 0,C 180,E1 -4747.097,E2 -4747.097} C_VEL
LIN {X 0,Y 523.619,Z 287.358,A -85,B 0,C 180,E1 -4749.978,E2 -4749.978} C_VEL
LIN {X 0,Y 523.497,Z 293.664,A -85,B 0,C 180,E1 -4752.822,E2 -4752.822} C_VEL
LIN {X 0,Y 523.446,Z 300.85,A -85,B 0,C 180,E1 -4756.015,E2 -4756.015} C_VEL
LIN {X 0,Y 523.426,Z 301.524,A -85,B 0,C 180,E1 -4756.311,E2 -4756.311} C_VEL
LIN {X 0,Y 525.393,Z 313.777,A -85,B 0,C 180,E1 -4756.659,E2 -4756.659} C_VEL
LIN {X 0,Y 525.127,Z 326.165,A -85,B 0,C 180,E1 -4757.095,E2 -4757.095} C_VEL
LIN {X 0,Y 524.816,Z 338.377,A -85,B 0,C 180,E1 -4757.695,E2 -4757.695} C_VEL
LIN {X 0,Y 524.611,Z 348.467,A -85,B 0,C 180,E1 -4758.333,E2 -4758.333} C_VEL
LIN {X 0,Y 524.366,Z 358.195,A -85,B 0,C 180,E1 -4759.087,E2 -4759.087} C_VEL
LIN {X 0,Y 524.084,Z 367.471,A -85,B 0,C 180,E1 -4759.96,E2 -4759.96} C_VEL
LIN {X 0,Y 523.901,Z 375.984,A -85,B 0,C 180,E1 -4760.931,E2 -4760.931} C_VEL
LIN {X 0,Y 523.692,Z 384.253,A -85,B 0,C 180,E1 -4762.094,E2 -4762.094} C_VEL
LIN {X 0,Y 523.58,Z 389.877,A -85,B 0,C 180,E1 -4763.061,E2 -4763.061} C_VEL
LIN {X 0,Y 523.52,Z 395.363,A -85,B 0,C 180,E1 -4764.222,E2 -4764.222} C_VEL
LIN {X 0,Y 523.361,Z 399.653,A -85,B 0,C 180,E1 -4765.379,E2 -4765.379} C_VEL
LIN {X 0,Y 523.445,Z 401.973,A -85,B 0,C 180,E1 -4766.151,E2 -4766.151} C_VEL
LIN {X 0,Y 523.369,Z 403.78,A -85,B 0,C 180,E1 -4766.921,E2 -4766.921} C_VEL
LIN {X 0,Y 523.276,Z 406.194,A -85,B 0,C 180,E1 -4768.461,E2 -4768.461} C_VEL
LIN {X 0,Y 523.251,Z 406.781,A -85,B 0,C 180,E1 -4769.23,E2 -4769.23} C_VEL
LIN {X 0,Y 523.251,Z 406.781,A -85,B 0,C 180,E1 -4770.77,E2 -4770.77} C_VEL
LIN {X 0,Y 523.276,Z 406.194,A -85,B 0,C 180,E1 -4771.539,E2 -4771.539} C_VEL
LIN {X 0,Y 523.369,Z 403.78,A -85,B 0,C 180,E1 -4773.079,E2 -4773.079} C_VEL
LIN {X 0,Y 523.443,Z 400.861,A -85,B 0,C 180,E1 -4774.235,E2 -4774.235} C_VEL
LIN {X 0,Y 523.464,Z 396.908,A -85,B 0,C 180,E1 -4775.393,E2 -4775.393} C_VEL
LIN {X 0,Y 523.521,Z 391.712,A -85,B 0,C 180,E1 -4776.572,E2 -4776.572} C_VEL
LIN {X 0,Y 523.669,Z 385.429,A -85,B 0,C 180,E1 -4777.713,E2 -4777.713} C_VEL
LIN {X 0,Y 523.858,Z 377.499,A -85,B 0,C 180,E1 -4778.875,E2 -4778.875} C_VEL
LIN {X 0,Y 524.083,Z 369.358,A -85,B 0,C 180,E1 -4779.845,E2 -4779.845} C_VEL
LIN {X 0,Y 524.334,Z 359.326,A -85,B 0,C 180,E1 -4780.816,E2 -4780.816} C_VEL
LIN {X 0,Y 524.613,Z 349.501,A -85,B 0,C 180,E1 -4781.592,E2 -4781.592} C_VEL
LIN {X 0,Y 524.793,Z 339.468,A -85,B 0,C 180,E1 -4782.24,E2 -4782.24} C_VEL
LIN {X 0,Y 525.108,Z 327.288,A -85,B 0,C 180,E1 -4782.856,E2 -4782.856} C_VEL
LIN {X 0,Y 525.366,Z 314.65,A -85,B 0,C 180,E1 -4783.317,E2 -4783.317} C_VEL
LIN {X 0,Y 524.537,Z 308.02,A -85,B 0,C 180,E1 -4783.523,E2 -4783.523} C_VEL
LIN {X 0,Y 523.426,Z 301.524,A -85,B 0,C 180,E1 -4783.689,E2 -4783.689} C_VEL
LIN {X 0,Y 523.443,Z 297.257,A -85,B 0,C 180,E1 -4785.576,E2 -4785.576} C_VEL
LIN {X 0,Y 523.52,Z 291.868,A -85,B 0,C 180,E1 -4787.984,E2 -4787.984} C_VEL
LIN {X 0,Y 523.622,Z 286.478,A -85,B 0,C 180,E1 -4790.424,E2 -4790.424} C_VEL
LIN {X 0,Y 523.689,Z 281.089,A -85,B 0,C 180,E1 -4792.903,E2 -4792.903} C_VEL
LIN {X 0,Y 523.809,Z 274.538,A -85,B 0,C 180,E1 -4795.977,E2 -4795.977} C_VEL
LIN {X 0,Y 523.9,Z 268.526,A -85,B 0,C 180,E1 -4798.876,E2 -4798.876} C_VEL
LIN {X 0,Y 524.012,Z 263.252,A -85,B 0,C 180,E1 -4801.537,E2 -4801.537} C_VEL
LIN {X 0,Y 524.148,Z 258.039,A -85,B 0,C 180,E1 -4804.273,E2 -4804.273} C_VEL
LIN {X 0,Y 524.332,Z 252.994,A -85,B 0,C 180,E1 -4807.096,E2 -4807.096} C_VEL
LIN {X 0,Y 524.532,Z 248.131,A -85,B 0,C 180,E1 -4810.025,E2 -4810.025} C_VEL
LIN {X 0,Y 524.502,Z 244.961,A -85,B 0,C 180,E1 -4812.064,E2 -4812.064} C_VEL
LIN {X 0,Y 523.995,Z 241.273,A -85,B 0,C 180,E1 -4814.693,E2 -4814.693} C_VEL
LIN {X 0,Y 523.922,Z 240.725,A -85,B 0,C 180,E1 -4815.311,E2 -4815.311} C_VEL
LIN {X 0,Y 523.917,Z 240.726,A -85,B 0,C 180,E1 -4818.693,E2 -4818.693} C_VEL
LIN {X 0,Y 523.915,Z 240.721,A -85,B 0,C 180,E1 -4821.895,E2 -4821.895} C_VEL
LIN {X 0,Y 523.92,Z 240.726,A -85,B 0,C 180,E1 -4824.91,E2 -4824.91} C_VEL
LIN {X 0,Y 523.935,Z 240.716,A -85,B 0,C 180,E1 -4827.678,E2 -4827.678} C_VEL
LIN {X 0,Y 523.94,Z 240.723,A -85,B 0,C 180,E1 -4830.678,E2 -4830.678} C_VEL
LIN {X 0,Y 523.902,Z 240.721,A -85,B 0,C 180,E1 -4833.721,E2 -4833.721} C_VEL
LIN {X 0,Y 523.91,Z 240.727,A -85,B 0,C 180,E1 -4836.266,E2 -4836.266} C_VEL
LIN {X 0,Y 523.933,Z 240.719,A -85,B 0,C 180,E1 -4838.763,E2 -4838.763} C_VEL
LIN {X 0,Y 523.926,Z 240.717,A -85,B 0,C 180,E1 -4841.216,E2 -4841.216} C_VEL
LIN {X 0,Y 523.911,Z 240.724,A -85,B 0,C 180,E1 -4844.434,E2 -4844.434} C_VEL
LIN {X 0,Y 523.958,Z 240.716,A -85,B 0,C 180,E1 -4847.603,E2 -4847.603} C_VEL
LIN {X 0,Y 523.927,Z 240.726,A -85,B 0,C 180,E1 -4849.953,E2 -4849.953} C_VEL
LIN {X 0,Y 523.987,Z 240.71,A -85,B 0,C 180,E1 -4853.063,E2 -4853.063} C_VEL
LIN {X 0,Y 523.944,Z 240.718,A -85,B 0,C 180,E1 -4855.38,E2 -4855.38} C_VEL
LIN {X 0,Y 524.094,Z 240.705,A -85,B 0,C 180,E1 -4857.69,E2 -4857.69} C_VEL
LIN {X 0,Y 524.084,Z 240.702,A -85,B 0,C 180,E1 -4859.996,E2 -4859.996} C_VEL
LIN {X 0,Y 524.026,Z 240.707,A -85,B 0,C 180,E1 -4863.071,E2 -4863.071} C_VEL
LIN {X 0,Y 524.002,Z 240.709,A -85,B 0,C 180,E1 -4866.155,E2 -4866.155} C_VEL
LIN {X 0,Y 523.964,Z 240.719,A -85,B 0,C 180,E1 -4869.257,E2 -4869.257} C_VEL
LIN {X 0,Y 523.982,Z 240.714,A -85,B 0,C 180,E1 -4871.733,E2 -4871.733} C_VEL
LIN {X 0,Y 523.961,Z 240.719,A -85,B 0,C 180,E1 -4875.043,E2 -4875.043} C_VEL
LIN {X 0,Y 523.921,Z 240.718,A -85,B 0,C 180,E1 -4877.965,E2 -4877.965} C_VEL
LIN {X 0,Y 523.932,Z 240.718,A -85,B 0,C 180,E1 -4880.406,E2 -4880.406} C_VEL
LIN {X 0,Y 523.882,Z 240.73,A -85,B 0,C 180,E1 -4882.889,E2 -4882.889} C_VEL
LIN {X 0,Y 523.952,Z 240.714,A -85,B 0,C 180,E1 -4886.014,E2 -4886.014} C_VEL
LIN {X 0,Y 523.906,Z 240.728,A -85,B 0,C 180,E1 -4888.87,E2 -4888.87} C_VEL
LIN {X 0,Y 523.884,Z 240.723,A -85,B 0,C 180,E1 -4891.539,E2 -4891.539} C_VEL
LIN {X 0,Y 523.905,Z 240.724,A -85,B 0,C 180,E1 -4894.285,E2 -4894.285} C_VEL
LIN {X 0,Y 523.87,Z 240.726,A -85,B 0,C 180,E1 -4897.127,E2 -4897.127} C_VEL
LIN {X 0,Y 523.894,Z 240.725,A -85,B 0,C 180,E1 -4900.125,E2 -4900.125} C_VEL
LIN {X 0,Y 523.894,Z 240.73,A -85,B 0,C 180,E1 -4902.455,E2 -4902.455} C_VEL
LIN {X 0,Y 523.906,Z 240.72,A -85,B 0,C 180,E1 -4905.304,E2 -4905.304} C_VEL
LIN {X 0,Y 523.872,Z 240.726,A -85,B 0,C 180,E1 -4906.872,E2 -4906.872} C_VEL
LIN {X 0,Y 523.196,Z 240.809,A -85,B 0,C 180,E1 -4907.514,E2 -4907.514} C_VEL
LIN {X 0,Y 520.334,Z 241.169,A -85,B 0,C 180,E1 -4908.555,E2 -4908.555} C_VEL
LIN {X 0,Y 517.935,Z 241.466,A -85,B 0,C 180,E1 -4909.394,E2 -4909.394} C_VEL
LIN {X 0,Y 516.927,Z 241.596,A -85,B 0,C 180,E1 -4910.042,E2 -4910.042} C_VEL
LIN {X 0,Y 516.858,Z 241.605,A -85,B 0,C 180,E1 -4910.261,E2 -4910.261} C_VEL
LIN {X 0,Y 516.829,Z 241.602,A -85,B 0,C 180,E1 -4913.338,E2 -4913.338} C_VEL
LIN {X 0,Y 516.856,Z 241.606,A -85,B 0,C 180,E1 -4916.118,E2 -4916.118} C_VEL
LIN {X 0,Y 516.847,Z 241.599,A -85,B 0,C 180,E1 -4918.929,E2 -4918.929} C_VEL
LIN {X 0,Y 516.864,Z 241.602,A -85,B 0,C 180,E1 -4921.582,E2 -4921.582} C_VEL
LIN {X 0,Y 516.884,Z 241.598,A -85,B 0,C 180,E1 -4924.209,E2 -4924.209} C_VEL
LIN {X 0,Y 516.847,Z 241.599,A -85,B 0,C 180,E1 -4926.776,E2 -4926.776} C_VEL
LIN {X 0,Y 516.874,Z 241.604,A -85,B 0,C 180,E1 -4929.729,E2 -4929.729} C_VEL
LIN {X 0,Y 516.877,Z 241.598,A -85,B 0,C 180,E1 -4932.595,E2 -4932.595} C_VEL
LIN {X 0,Y 516.897,Z 241.598,A -85,B 0,C 180,E1 -4935.029,E2 -4935.029} C_VEL
LIN {X 0,Y 516.935,Z 241.59,A -85,B 0,C 180,E1 -4938.233,E2 -4938.233} C_VEL
LIN {X 0,Y 516.91,Z 241.599,A -85,B 0,C 180,E1 -4941.399,E2 -4941.399} C_VEL
LIN {X 0,Y 516.954,Z 241.59,A -85,B 0,C 180,E1 -4943.756,E2 -4943.756} C_VEL
LIN {X 0,Y 516.981,Z 241.59,A -85,B 0,C 180,E1 -4946.883,E2 -4946.883} C_VEL
LIN {X 0,Y 517.013,Z 241.581,A -85,B 0,C 180,E1 -4950,E2 -4950} C_VEL
LIN {X 0,Y 516.981,Z 241.59,A -85,B 0,C 180,E1 -4953.117,E2 -4953.117} C_VEL
LIN {X 0,Y 516.954,Z 241.59,A -85,B 0,C 180,E1 -4956.244,E2 -4956.244} C_VEL
LIN {X 0,Y 516.91,Z 241.599,A -85,B 0,C 180,E1 -4958.601,E2 -4958.601} C_VEL
LIN {X 0,Y 516.915,Z 241.593,A -85,B 0,C 180,E1 -4961.825,E2 -4961.825} C_VEL
LIN {X 0,Y 516.891,Z 241.597,A -85,B 0,C 180,E1 -4965.154,E2 -4965.154} C_VEL
LIN {X 0,Y 516.865,Z 241.604,A -85,B 0,C 180,E1 -4968.224,E2 -4968.224} C_VEL
LIN {X 0,Y 516.852,Z 241.603,A -85,B 0,C 180,E1 -4970.704,E2 -4970.704} C_VEL
LIN {X 0,Y 516.847,Z 241.599,A -85,B 0,C 180,E1 -4973.224,E2 -4973.224} C_VEL
LIN {X 0,Y 516.886,Z 241.603,A -85,B 0,C 180,E1 -4976.201,E2 -4976.201} C_VEL
LIN {X 0,Y 516.876,Z 241.596,A -85,B 0,C 180,E1 -4979.307,E2 -4979.307} C_VEL
LIN {X 0,Y 516.844,Z 241.602,A -85,B 0,C 180,E1 -4982.548,E2 -4982.548} C_VEL
LIN {X 0,Y 516.827,Z 241.603,A -85,B 0,C 180,E1 -4985.336,E2 -4985.336} C_VEL
LIN {X 0,Y 516.828,Z 241.61,A -85,B 0,C 180,E1 -4987.947,E2 -4987.947} C_VEL
LIN {X 0,Y 516.852,Z 241.599,A -85,B 0,C 180,E1 -4990.744,E2 -4990.744} C_VEL
LIN {X 0,Y 516.833,Z 241.607,A -85,B 0,C 180,E1 -4993.907,E2 -4993.907} C_VEL
LIN {X 0,Y 516.835,Z 241.603,A -85,B 0,C 180,E1 -4996.111,E2 -4996.111} C_VEL
LIN {X 0,Y 516.877,Z 241.596,A -85,B 0,C 180,E1 -4998.402,E2 -4998.402} C_VEL
LIN {X 0,Y 516.837,Z 241.607,A -85,B 0,C 180,E1 -5001.289,E2 -5001.289} C_VEL
LIN {X 0,Y 516.85,Z 241.599,A -85,B 0,C 180,E1 -5004.226,E2 -5004.226} C_VEL
LIN {X 0,Y 516.857,Z 241.603,A -85,B 0,C 180,E1 -5007.058,E2 -5007.058} C_VEL
LIN {X 0,Y 516.856,Z 241.6,A -85,B 0,C 180,E1 -5009.801,E2 -5009.801} C_VEL
LIN {X 0,Y 516.896,Z 241.594,A -85,B 0,C 180,E1 -5012.472,E2 -5012.472} C_VEL
LIN {X 0,Y 516.87,Z 241.605,A -85,B 0,C 180,E1 -5015.076,E2 -5015.076} C_VEL
LIN {X 0,Y 516.858,Z 241.6,A -85,B 0,C 180,E1 -5018.467,E2 -5018.467} C_VEL
LIN {X 0,Y 516.868,Z 241.605,A -85,B 0,C 180,E1 -5020.96,E2 -5020.96} C_VEL
LIN {X 0,Y 516.878,Z 241.597,A -85,B 0,C 180,E1 -5023.415,E2 -5023.415} C_VEL
LIN {X 0,Y 516.853,Z 241.599,A -85,B 0,C 180,E1 -5025.838,E2 -5025.838} C_VEL
LIN {X 0,Y 516.948,Z 241.59,A -85,B 0,C 180,E1 -5028.239,E2 -5028.239} C_VEL
LIN {X 0,Y 516.936,Z 241.588,A -85,B 0,C 180,E1 -5031.404,E2 -5031.404} C_VEL
LIN {X 0,Y 516.97,Z 241.585,A -85,B 0,C 180,E1 -5033.761,E2 -5033.761} C_VEL
LIN {X 0,Y 516.969,Z 241.587,A -85,B 0,C 180,E1 -5036.888,E2 -5036.888} C_VEL
LIN {X 0,Y 516.953,Z 241.594,A -85,B 0,C 180,E1 -5038.447,E2 -5038.447} C_VEL
LIN {X 0,Y 517.08,Z 241.573,A -85,B 0,C 180,E1 -5040.783,E2 -5040.783} C_VEL
LIN {X 0,Y 516.938,Z 241.588,A -85,B 0,C 180,E1 -5043.122,E2 -5043.122} C_VEL
LIN {X 0,Y 516.966,Z 241.592,A -85,B 0,C 180,E1 -5046.248,E2 -5046.248} C_VEL
LIN {X 0,Y 516.931,Z 241.59,A -85,B 0,C 180,E1 -5049.394,E2 -5049.394} C_VEL
LIN {X 0,Y 516.951,Z 241.593,A -85,B 0,C 180,E1 -5051.811,E2 -5051.811} C_VEL
LIN {X 0,Y 516.939,Z 241.589,A -85,B 0,C 180,E1 -5055.147,E2 -5055.147} C_VEL
LIN {X 0,Y 516.875,Z 241.599,A -85,B 0,C 180,E1 -5058.228,E2 -5058.228} C_VEL
LIN {X 0,Y 516.896,Z 241.593,A -85,B 0,C 180,E1 -5060.706,E2 -5060.706} C_VEL
LIN {X 0,Y 516.858,Z 241.601,A -85,B 0,C 180,E1 -5063.228,E2 -5063.228} C_VEL
LIN {X 0,Y 516.882,Z 241.596,A -85,B 0,C 180,E1 -5066.184,E2 -5066.184} C_VEL
LIN {X 0,Y 516.89,Z 241.602,A -85,B 0,C 180,E1 -5069.521,E2 -5069.521} C_VEL
LIN {X 0,Y 516.897,Z 241.594,A -85,B 0,C 180,E1 -5072.545,E2 -5072.545} C_VEL
LIN {X 0,Y 516.859,Z 241.606,A -85,B 0,C 180,E1 -5075.33,E2 -5075.33} C_VEL
LIN {X 0,Y 516.881,Z 241.598,A -85,B 0,C 180,E1 -5077.944,E2 -5077.944} C_VEL
LIN {X 0,Y 516.858,Z 241.605,A -85,B 0,C 180,E1 -5080.747,E2 -5080.747} C_VEL
LIN {X 0,Y 516.867,Z 241.604,A -85,B 0,C 180,E1 -5083.908,E2 -5083.908} C_VEL
LIN {X 0,Y 516.966,Z 242.167,A -85,B 0,C 180,E1 -5085.016,E2 -5085.016} C_VEL
LIN {X 0,Y 517.366,Z 245.192,A -85,B 0,C 180,E1 -5087.219,E2 -5087.219} C_VEL
LIN {X 0,Y 517.575,Z 248.318,A -85,B 0,C 180,E1 -5089.325,E2 -5089.325} C_VEL
LIN {X 0,Y 517.414,Z 253.159,A -85,B 0,C 180,E1 -5092.322,E2 -5092.322} C_VEL
LIN {X 0,Y 517.15,Z 258.156,A -85,B 0,C 180,E1 -5095.196,E2 -5095.196} C_VEL
LIN {X 0,Y 517.018,Z 263.329,A -85,B 0,C 180,E1 -5097.986,E2 -5097.986} C_VEL
LIN {X 0,Y 516.914,Z 268.592,A -85,B 0,C 180,E1 -5100.696,E2 -5100.696} C_VEL
LIN {X 0,Y 516.748,Z 274.973,A -85,B 0,C 180,E1 -5103.851,E2 -5103.851} C_VEL
LIN {X 0,Y 516.61,Z 281.089,A -85,B 0,C 180,E1 -5106.765,E2 -5106.765} C_VEL
LIN {X 0,Y 516.556,Z 287.703,A -85,B 0,C 180,E1 -5109.851,E2 -5109.851} C_VEL
LIN {X 0,Y 516.436,Z 293.664,A -85,B 0,C 180,E1 -5112.579,E2 -5112.579} C_VEL
LIN {X 0,Y 516.363,Z 300.85,A -85,B 0,C 180,E1 -5115.819,E2 -5115.819} C_VEL
LIN {X 0,Y 516.382,Z 301.524,A -85,B 0,C 180,E1 -5116.121,E2 -5116.121} C_VEL
LIN {X 0,Y 518.457,Z 313.761,A -85,B 0,C 180,E1 -5116.477,E2 -5116.477} C_VEL
LIN {X 0,Y 518.21,Z 326.166,A -85,B 0,C 180,E1 -5116.92,E2 -5116.92} C_VEL
LIN {X 0,Y 517.86,Z 338.501,A -85,B 0,C 180,E1 -5117.535,E2 -5117.535} C_VEL
LIN {X 0,Y 517.683,Z 347.823,A -85,B 0,C 180,E1 -5118.127,E2 -5118.127} C_VEL
LIN {X 0,Y 517.381,Z 358.188,A -85,B 0,C 180,E1 -5118.938,E2 -5118.938} C_VEL
LIN {X 0,Y 517.16,Z 365.553,A -85,B 0,C 180,E1 -5119.627,E2 -5119.627} C_VEL
LIN {X 0,Y 516.954,Z 372.739,A -85,B 0,C 180,E1 -5120.414,E2 -5120.414} C_VEL
LIN {X 0,Y 516.756,Z 380.284,A -85,B 0,C 180,E1 -5121.396,E2 -5121.396} C_VEL
LIN {X 0,Y 516.567,Z 386.574,A -85,B 0,C 180,E1 -5122.377,E2 -5122.377} C_VEL
LIN {X 0,Y 516.447,Z 392.145,A -85,B 0,C 180,E1 -5123.427,E2 -5123.427} C_VEL
LIN {X 0,Y 516.402,Z 396.904,A -85,B 0,C 180,E1 -5124.533,E2 -5124.533} C_VEL
LIN {X 0,Y 516.345,Z 400.858,A -85,B 0,C 180,E1 -5125.707,E2 -5125.707} C_VEL
LIN {X 0,Y 516.285,Z 403.777,A -85,B 0,C 180,E1 -5126.879,E2 -5126.879} C_VEL
LIN {X 0,Y 516.193,Z 406.195,A -85,B 0,C 180,E1 -5128.44,E2 -5128.44} C_VEL
LIN {X 0,Y 516.161,Z 406.78,A -85,B 0,C 180,E1 -5129.22,E2 -5129.22} C_VEL
LIN {X 0,Y 516.161,Z 406.78,A -85,B 0,C 180,E1 -5130.78,E2 -5130.78} C_VEL
LIN {X 0,Y 516.193,Z 406.195,A -85,B 0,C 180,E1 -5131.56,E2 -5131.56} C_VEL
LIN {X 0,Y 516.285,Z 403.777,A -85,B 0,C 180,E1 -5133.121,E2 -5133.121} C_VEL
LIN {X 0,Y 516.345,Z 400.858,A -85,B 0,C 180,E1 -5134.293,E2 -5134.293} C_VEL
LIN {X 0,Y 516.402,Z 396.904,A -85,B 0,C 180,E1 -5135.467,E2 -5135.467} C_VEL
LIN {X 0,Y 516.448,Z 392.144,A -85,B 0,C 180,E1 -5136.573,E2 -5136.573} C_VEL
LIN {X 0,Y 516.567,Z 386.574,A -85,B 0,C 180,E1 -5137.623,E2 -5137.623} C_VEL
LIN {X 0,Y 516.756,Z 380.284,A -85,B 0,C 180,E1 -5138.604,E2 -5138.604} C_VEL
LIN {X 0,Y 516.954,Z 372.739,A -85,B 0,C 180,E1 -5139.586,E2 -5139.586} C_VEL
LIN {X 0,Y 517.231,Z 363.626,A -85,B 0,C 180,E1 -5140.57,E2 -5140.57} C_VEL
LIN {X 0,Y 517.561,Z 352.19,A -85,B 0,C 180,E1 -5141.554,E2 -5141.554} C_VEL
LIN {X 0,Y 517.749,Z 342.627,A -85,B 0,C 180,E1 -5142.216,E2 -5142.216} C_VEL
LIN {X 0,Y 518.037,Z 331.409,A -85,B 0,C 180,E1 -5142.835,E2 -5142.835} C_VEL
LIN {X 0,Y 518.286,Z 321.065,A -85,B 0,C 180,E1 -5143.278,E2 -5143.278} C_VEL
LIN {X 0,Y 518.319,Z 312.887,A -85,B 0,C 180,E1 -5143.551,E2 -5143.551} C_VEL
LIN {X 0,Y 516.382,Z 301.524,A -85,B 0,C 180,E1 -5143.879,E2 -5143.879} C_VEL
LIN {X 0,Y 516.374,Z 295.461,A -85,B 0,C 180,E1 -5146.607,E2 -5146.607} C_VEL
LIN {X 0,Y 516.465,Z 290.071,A -85,B 0,C 180,E1 -5149.062,E2 -5149.062} C_VEL
LIN {X 0,Y 516.556,Z 284.682,A -85,B 0,C 180,E1 -5151.552,E2 -5151.552} C_VEL
LIN {X 0,Y 516.677,Z 278.829,A -85,B 0,C 180,E1 -5154.304,E2 -5154.304} C_VEL
LIN {X 0,Y 516.812,Z 272.1,A -85,B 0,C 180,E1 -5157.539,E2 -5157.539} C_VEL
LIN {X 0,Y 516.931,Z 266.838,A -85,B 0,C 180,E1 -5160.201,E2 -5160.201} C_VEL
LIN {X 0,Y 517.058,Z 261.575,A -85,B 0,C 180,E1 -5162.935,E2 -5162.935} C_VEL
LIN {X 0,Y 517.21,Z 256.453,A -85,B 0,C 180,E1 -5165.753,E2 -5165.753} C_VEL
LIN {X 0,Y 517.469,Z 251.512,A -85,B 0,C 180,E1 -5168.663,E2 -5168.663} C_VEL
LIN {X 0,Y 517.578,Z 246.731,A -85,B 0,C 180,E1 -5171.708,E2 -5171.708} C_VEL
LIN {X 0,Y 517.176,Z 243.587,A -85,B 0,C 180,E1 -5173.924,E2 -5173.924} C_VEL
LIN {X 0,Y 516.966,Z 242.12,A -85,B 0,C 180,E1 -5175.012,E2 -5175.012} C_VEL
LIN {X 0,Y 516.867,Z 241.602,A -85,B 0,C 180,E1 -5176.108,E2 -5176.108} C_VEL
LIN {X 0,Y 516.853,Z 241.605,A -85,B 0,C 180,E1 -5179.252,E2 -5179.252} C_VEL
LIN {X 0,Y 516.881,Z 241.598,A -85,B 0,C 180,E1 -5182.056,E2 -5182.056} C_VEL
LIN {X 0,Y 516.876,Z 241.599,A -85,B 0,C 180,E1 -5185.172,E2 -5185.172} C_VEL
LIN {X 0,Y 516.872,Z 241.597,A -85,B 0,C 180,E1 -5187.972,E2 -5187.972} C_VEL
LIN {X 0,Y 516.907,Z 241.599,A -85,B 0,C 180,E1 -5190.691,E2 -5190.691} C_VEL
LIN {X 0,Y 516.882,Z 241.596,A -85,B 0,C 180,E1 -5193.816,E2 -5193.816} C_VEL
LIN {X 0,Y 516.858,Z 241.601,A -85,B 0,C 180,E1 -5196.772,E2 -5196.772} C_VEL
LIN {X 0,Y 516.909,Z 241.593,A -85,B 0,C 180,E1 -5199.738,E2 -5199.738} C_VEL
LIN {X 0,Y 516.866,Z 241.6,A -85,B 0,C 180,E1 -5202.59,E2 -5202.59} C_VEL
LIN {X 0,Y 516.935,Z 241.589,A -85,B 0,C 180,E1 -5205.026,E2 -5205.026} C_VEL
LIN {X 0,Y 516.965,Z 241.591,A -85,B 0,C 180,E1 -5208.23,E2 -5208.23} C_VEL
LIN {X 0,Y 516.926,Z 241.591,A -85,B 0,C 180,E1 -5211.395,E2 -5211.395} C_VEL
LIN {X 0,Y 516.979,Z 241.584,A -85,B 0,C 180,E1 -5214.535,E2 -5214.535} C_VEL
LIN {X 0,Y 517.064,Z 241.58,A -85,B 0,C 180,E1 -5217.659,E2 -5217.659} C_VEL
LIN {X 0,Y 517.053,Z 241.578,A -85,B 0,C 180,E1 -5219.995,E2 -5219.995} C_VEL
LIN {X 0,Y 517.063,Z 241.573,A -85,B 0,C 180,E1 -5222.332,E2 -5222.332} C_VEL
LIN {X 0,Y 516.999,Z 241.588,A -85,B 0,C 180,E1 -5225.455,E2 -5225.455} C_VEL
LIN {X 0,Y 516.946,Z 241.591,A -85,B 0,C 180,E1 -5227.809,E2 -5227.809} C_VEL
LIN {X 0,Y 516.932,Z 241.592,A -85,B 0,C 180,E1 -5230.967,E2 -5230.967} C_VEL
LIN {X 0,Y 516.882,Z 241.603,A -85,B 0,C 180,E1 -5233.359,E2 -5233.359} C_VEL
LIN {X 0,Y 516.875,Z 241.598,A -85,B 0,C 180,E1 -5235.774,E2 -5235.774} C_VEL
LIN {X 0,Y 516.889,Z 241.594,A -85,B 0,C 180,E1 -5238.218,E2 -5238.218} C_VEL
LIN {X 0,Y 516.878,Z 241.599,A -85,B 0,C 180,E1 -5240.697,E2 -5240.697} C_VEL
LIN {X 0,Y 516.86,Z 241.598,A -85,B 0,C 180,E1 -5244.068,E2 -5244.068} C_VEL
LIN {X 0,Y 516.894,Z 241.599,A -85,B 0,C 180,E1 -5246.653,E2 -5246.653} C_VEL
LIN {X 0,Y 516.876,Z 241.596,A -85,B 0,C 180,E1 -5249.519,E2 -5249.519} C_VEL
LIN {X 0,Y 516.858,Z 241.604,A -85,B 0,C 180,E1 -5252.538,E2 -5252.538} C_VEL
LIN {X 0,Y 516.843,Z 241.601,A -85,B 0,C 180,E1 -5255.327,E2 -5255.327} C_VEL
LIN {X 0,Y 516.838,Z 241.602,A -85,B 0,C 180,E1 -5257.938,E2 -5257.938} C_VEL
LIN {X 0,Y 516.85,Z 241.604,A -85,B 0,C 180,E1 -5260.736,E2 -5260.736} C_VEL
LIN {X 0,Y 516.858,Z 241.601,A -85,B 0,C 180,E1 -5262.825,E2 -5262.825} C_VEL
LIN {X 0,Y 516.874,Z 241.597,A -85,B 0,C 180,E1 -5265.006,E2 -5265.006} C_VEL
LIN {X 0,Y 516.872,Z 241.603,A -85,B 0,C 180,E1 -5268.393,E2 -5268.393} C_VEL
LIN {X 0,Y 516.858,Z 241.605,A -85,B 0,C 180,E1 -5270.261,E2 -5270.261} C_VEL
LIN {X 0,Y 516.221,Z 241.692,A -85,B 0,C 180,E1 -5270.911,E2 -5270.911} C_VEL
LIN {X 0,Y 513.367,Z 242.048,A -85,B 0,C 180,E1 -5271.966,E2 -5271.966} C_VEL
LIN {X 0,Y 510.927,Z 242.346,A -85,B 0,C 180,E1 -5272.816,E2 -5272.816} C_VEL
LIN {X 0,Y 509.868,Z 242.473,A -85,B 0,C 180,E1 -5273.473,E2 -5273.473} C_VEL
LIN {X 0,Y 509.777,Z 242.483,A -85,B 0,C 180,E1 -5273.695,E2 -5273.695} C_VEL
LIN {X 0,Y 509.806,Z 242.478,A -85,B 0,C 180,E1 -5276.536,E2 -5276.536} C_VEL
LIN {X 0,Y 509.803,Z 242.478,A -85,B 0,C 180,E1 -5279.332,E2 -5279.332} C_VEL
LIN {X 0,Y 509.835,Z 242.478,A -85,B 0,C 180,E1 -5282.052,E2 -5282.052} C_VEL
LIN {X 0,Y 509.837,Z 242.473,A -85,B 0,C 180,E1 -5284.702,E2 -5284.702} C_VEL
LIN {X 0,Y 509.82,Z 242.48,A -85,B 0,C 180,E1 -5287.44,E2 -5287.44} C_VEL
LIN {X 0,Y 509.852,Z 242.478,A -85,B 0,C 180,E1 -5289.842,E2 -5289.842} C_VEL
LIN {X 0,Y 509.838,Z 242.479,A -85,B 0,C 180,E1 -5293.174,E2 -5293.174} C_VEL
LIN {X 0,Y 509.817,Z 242.482,A -85,B 0,C 180,E1 -5295.633,E2 -5295.633} C_VEL
LIN {X 0,Y 509.875,Z 242.47,A -85,B 0,C 180,E1 -5298.099,E2 -5298.099} C_VEL
LIN {X 0,Y 509.884,Z 242.476,A -85,B 0,C 180,E1 -5301.279,E2 -5301.279} C_VEL
LIN {X 0,Y 509.924,Z 242.466,A -85,B 0,C 180,E1 -5303.67,E2 -5303.67} C_VEL
LIN {X 0,Y 509.922,Z 242.47,A -85,B 0,C 180,E1 -5306.84,E2 -5306.84} C_VEL
LIN {X 0,Y 509.984,Z 242.457,A -85,B 0,C 180,E1 -5310,E2 -5310} C_VEL
LIN {X 0,Y 509.922,Z 242.47,A -85,B 0,C 180,E1 -5313.16,E2 -5313.16} C_VEL
LIN {X 0,Y 509.924,Z 242.466,A -85,B 0,C 180,E1 -5316.33,E2 -5316.33} C_VEL
LIN {X 0,Y 509.884,Z 242.476,A -85,B 0,C 180,E1 -5318.721,E2 -5318.721} C_VEL
LIN {X 0,Y 509.884,Z 242.469,A -85,B 0,C 180,E1 -5321.932,E2 -5321.932} C_VEL
LIN {X 0,Y 509.856,Z 242.473,A -85,B 0,C 180,E1 -5325.256,E2 -5325.256} C_VEL
LIN {X 0,Y 509.845,Z 242.476,A -85,B 0,C 180,E1 -5328.011,E2 -5328.011} C_VEL
LIN {X 0,Y 509.797,Z 242.479,A -85,B 0,C 180,E1 -5331.004,E2 -5331.004} C_VEL
LIN {X 0,Y 509.806,Z 242.477,A -85,B 0,C 180,E1 -5333.564,E2 -5333.564} C_VEL
LIN {X 0,Y 509.855,Z 242.477,A -85,B 0,C 180,E1 -5336.383,E2 -5336.383} C_VEL
LIN {X 0,Y 509.825,Z 242.475,A -85,B 0,C 180,E1 -5338.847,E2 -5338.847} C_VEL
LIN {X 0,Y 509.774,Z 242.483,A -85,B 0,C 180,E1 -5341.593,E2 -5341.593} C_VEL
LIN {X 0,Y 509.798,Z 242.48,A -85,B 0,C 180,E1 -5344.417,E2 -5344.417} C_VEL
LIN {X 0,Y 509.764,Z 242.484,A -85,B 0,C 180,E1 -5347.344,E2 -5347.344} C_VEL
LIN {X 0,Y 509.809,Z 242.478,A -85,B 0,C 180,E1 -5350.384,E2 -5350.384} C_VEL
LIN {X 0,Y 509.789,Z 242.48,A -85,B 0,C 180,E1 -5353.069,E2 -5353.069} C_VEL
LIN {X 0,Y 509.783,Z 242.486,A -85,B 0,C 180,E1 -5355.797,E2 -5355.797} C_VEL
LIN {X 0,Y 509.819,Z 242.475,A -85,B 0,C 180,E1 -5358.58,E2 -5358.58} C_VEL
LIN {X 0,Y 509.808,Z 242.48,A -85,B 0,C 180,E1 -5361.791,E2 -5361.791} C_VEL
LIN {X 0,Y 509.806,Z 242.477,A -85,B 0,C 180,E1 -5364.628,E2 -5364.628} C_VEL
LIN {X 0,Y 509.823,Z 242.48,A -85,B 0,C 180,E1 -5367.486,E2 -5367.486} C_VEL
LIN {X 0,Y 509.824,Z 242.474,A -85,B 0,C 180,E1 -5370.279,E2 -5370.279} C_VEL
LIN {X 0,Y 509.853,Z 242.477,A -85,B 0,C 180,E1 -5372.95,E2 -5372.95} C_VEL
LIN {X 0,Y 509.823,Z 242.476,A -85,B 0,C 180,E1 -5375.578,E2 -5375.578} C_VEL
LIN {X 0,Y 509.794,Z 242.478,A -85,B 0,C 180,E1 -5378.154,E2 -5378.154} C_VEL
LIN {X 0,Y 509.832,Z 242.479,A -85,B 0,C 180,E1 -5380.686,E2 -5380.686} C_VEL
LIN {X 0,Y 509.844,Z 242.475,A -85,B 0,C 180,E1 -5383.179,E2 -5383.179} C_VEL
LIN {X 0,Y 509.825,Z 242.474,A -85,B 0,C 180,E1 -5385.639,E2 -5385.639} C_VEL
LIN {X 0,Y 509.894,Z 242.471,A -85,B 0,C 180,E1 -5388.879,E2 -5388.879} C_VEL
LIN {X 0,Y 509.905,Z 242.467,A -85,B 0,C 180,E1 -5392.083,E2 -5392.083} C_VEL
LIN {X 0,Y 509.951,Z 242.467,A -85,B 0,C 180,E1 -5394.469,E2 -5394.469} C_VEL
LIN {X 0,Y 510.034,Z 242.449,A -85,B 0,C 180,E1 -5397.636,E2 -5397.636} C_VEL
LIN {X 0,Y 510.03,Z 242.451,A -85,B 0,C 180,E1 -5400.794,E2 -5400.794} C_VEL
LIN {X 0,Y 509.883,Z 242.467,A -85,B 0,C 180,E1 -5403.165,E2 -5403.165} C_VEL
LIN {X 0,Y 509.913,Z 242.469,A -85,B 0,C 180,E1 -5406.335,E2 -5406.335} C_VEL
LIN {X 0,Y 509.872,Z 242.47,A -85,B 0,C 180,E1 -5409.525,E2 -5409.525} C_VEL
LIN {X 0,Y 509.903,Z 242.473,A -85,B 0,C 180,E1 -5411.936,E2 -5411.936} C_VEL
LIN {X 0,Y 509.895,Z 242.467,A -85,B 0,C 180,E1 -5415.246,E2 -5415.246} C_VEL
LIN {X 0,Y 509.834,Z 242.474,A -85,B 0,C 180,E1 -5418.488,E2 -5418.488} C_VEL
LIN {X 0,Y 509.839,Z 242.473,A -85,B 0,C 180,E1 -5421.006,E2 -5421.006} C_VEL
LIN {X 0,Y 509.82,Z 242.483,A -85,B 0,C 180,E1 -5423.567,E2 -5423.567} C_VEL
LIN {X 0,Y 509.818,Z 242.475,A -85,B 0,C 180,E1 -5426.359,E2 -5426.359} C_VEL
LIN {X 0,Y 509.838,Z 242.474,A -85,B 0,C 180,E1 -5428.85,E2 -5428.85} C_VEL
LIN {X 0,Y 509.817,Z 242.481,A -85,B 0,C 180,E1 -5431.594,E2 -5431.594} C_VEL
LIN {X 0,Y 509.838,Z 242.474,A -85,B 0,C 180,E1 -5434.418,E2 -5434.418} C_VEL
LIN {X 0,Y 509.811,Z 242.484,A -85,B 0,C 180,E1 -5437.344,E2 -5437.344} C_VEL
LIN {X 0,Y 509.82,Z 242.479,A -85,B 0,C 180,E1 -5440.387,E2 -5440.387} C_VEL
LIN {X 0,Y 509.799,Z 242.484,A -85,B 0,C 180,E1 -5443.577,E2 -5443.577} C_VEL
LIN {X 0,Y 509.815,Z 242.483,A -85,B 0,C 180,E1 -5444.207,E2 -5444.207} C_VEL
LIN {X 0,Y 510.309,Z 245.956,A -85,B 0,C 180,E1 -5446.882,E2 -5446.882} C_VEL
LIN {X 0,Y 510.592,Z 249.335,A -85,B 0,C 180,E1 -5449.207,E2 -5449.207} C_VEL
LIN {X 0,Y 510.43,Z 253.277,A -85,B 0,C 180,E1 -5451.714,E2 -5451.714} C_VEL
LIN {X 0,Y 510.167,Z 258.259,A -85,B 0,C 180,E1 -5454.65,E2 -5454.65} C_VEL
LIN {X 0,Y 510.005,Z 263.338,A -85,B 0,C 180,E1 -5457.492,E2 -5457.492} C_VEL
LIN {X 0,Y 509.867,Z 268.637,A -85,B 0,C 180,E1 -5460.275,E2 -5460.275} C_VEL
LIN {X 0,Y 509.71,Z 275.356,A -85,B 0,C 180,E1 -5463.671,E2 -5463.671} C_VEL
LIN {X 0,Y 509.552,Z 281.089,A -85,B 0,C 180,E1 -5466.423,E2 -5466.423} C_VEL
LIN {X 0,Y 509.497,Z 288.046,A -85,B 0,C 180,E1 -5469.721,E2 -5469.721} C_VEL
LIN {X 0,Y 509.399,Z 293.664,A -85,B 0,C 180,E1 -5472.331,E2 -5472.331} C_VEL
LIN {X 0,Y 509.294,Z 301.299,A -85,B 0,C 180,E1 -5475.822,E2 -5475.822} C_VEL
LIN {X 0,Y 509.284,Z 301.524,A -85,B 0,C 180,E1 -5475.924,E2 -5475.924} C_VEL
LIN {X 0,Y 511.378,Z 313.745,A -85,B 0,C 180,E1 -5476.287,E2 -5476.287} C_VEL
LIN {X 0,Y 511.354,Z 323.628,A -85,B 0,C 180,E1 -5476.64,E2 -5476.64} C_VEL
LIN {X 0,Y 511.046,Z 335.397,A -85,B 0,C 180,E1 -5477.188,E2 -5477.188} C_VEL
LIN {X 0,Y 510.689,Z 346.917,A -85,B 0,C 180,E1 -5477.897,E2 -5477.897} C_VEL
LIN {X 0,Y 510.472,Z 357.05,A -85,B 0,C 180,E1 -5478.686,E2 -5478.686} C_VEL
LIN {X 0,Y 510.171,Z 365.547,A -85,B 0,C 180,E1 -5479.483,E2 -5479.483} C_VEL
LIN {X 0,Y 509.951,Z 372.734,A -85,B 0,C 180,E1 -5480.281,E2 -5480.281} C_VEL
LIN {X 0,Y 509.72,Z 380.28,A -85,B 0,C 180,E1 -5481.277,E2 -5481.277} C_VEL
LIN {X 0,Y 509.527,Z 386.569,A -85,B 0,C 180,E1 -5482.271,E2 -5482.271} C_VEL
LIN {X 0,Y 509.357,Z 392.657,A -85,B 0,C 180,E1 -5483.443,E2 -5483.443} C_VEL
LIN {X 0,Y 509.248,Z 398.386,A -85,B 0,C 180,E1 -5484.853,E2 -5484.853} C_VEL
LIN {X 0,Y 509.255,Z 401.975,A -85,B 0,C 180,E1 -5486.043,E2 -5486.043} C_VEL
LIN {X 0,Y 509.203,Z 403.775,A -85,B 0,C 180,E1 -5486.835,E2 -5486.835} C_VEL
LIN {X 0,Y 509.114,Z 406.195,A -85,B 0,C 180,E1 -5488.418,E2 -5488.418} C_VEL
LIN {X 0,Y 509.075,Z 406.78,A -85,B 0,C 180,E1 -5489.209,E2 -5489.209} C_VEL
LIN {X 0,Y 509.075,Z 406.78,A -85,B 0,C 180,E1 -5490.791,E2 -5490.791} C_VEL
LIN {X 0,Y 509.114,Z 406.195,A -85,B 0,C 180,E1 -5491.582,E2 -5491.582} C_VEL
LIN {X 0,Y 509.203,Z 403.775,A -85,B 0,C 180,E1 -5493.165,E2 -5493.165} C_VEL
LIN {X 0,Y 509.235,Z 400.854,A -85,B 0,C 180,E1 -5494.353,E2 -5494.353} C_VEL
LIN {X 0,Y 509.339,Z 396.899,A -85,B 0,C 180,E1 -5495.543,E2 -5495.543} C_VEL
LIN {X 0,Y 509.41,Z 391.278,A -85,B 0,C 180,E1 -5496.844,E2 -5496.844} C_VEL
LIN {X 0,Y 509.589,Z 384.255,A -85,B 0,C 180,E1 -5498.127,E2 -5498.127} C_VEL
LIN {X 0,Y 509.845,Z 375.976,A -85,B 0,C 180,E1 -5499.321,E2 -5499.321} C_VEL
LIN {X 0,Y 510.054,Z 367.46,A -85,B 0,C 180,E1 -5500.319,E2 -5500.319} C_VEL
LIN {X 0,Y 510.354,Z 359.313,A -85,B 0,C 180,E1 -5501.116,E2 -5501.116} C_VEL
LIN {X 0,Y 510.654,Z 350.834,A -85,B 0,C 180,E1 -5501.813,E2 -5501.813} C_VEL
LIN {X 0,Y 510.846,Z 340.905,A -85,B 0,C 180,E1 -5502.49,E2 -5502.49} C_VEL
LIN {X 0,Y 511.143,Z 330.394,A -85,B 0,C 180,E1 -5503.062,E2 -5503.062} C_VEL
LIN {X 0,Y 511.471,Z 318.476,A -85,B 0,C 180,E1 -5503.559,E2 -5503.559} C_VEL
LIN {X 0,Y 511.3,Z 313.308,A -85,B 0,C 180,E1 -5503.728,E2 -5503.728} C_VEL
LIN {X 0,Y 509.284,Z 301.524,A -85,B 0,C 180,E1 -5504.076,E2 -5504.076} C_VEL
LIN {X 0,Y 509.313,Z 295.461,A -85,B 0,C 180,E1 -5506.844,E2 -5506.844} C_VEL
LIN {X 0,Y 509.399,Z 290.071,A -85,B 0,C 180,E1 -5509.336,E2 -5509.336} C_VEL
LIN {X 0,Y 509.51,Z 284.682,A -85,B 0,C 180,E1 -5511.865,E2 -5511.865} C_VEL
LIN {X 0,Y 509.634,Z 279.226,A -85,B 0,C 180,E1 -5514.469,E2 -5514.469} C_VEL
LIN {X 0,Y 509.725,Z 273.851,A -85,B 0,C 180,E1 -5517.064,E2 -5517.064} C_VEL
LIN {X 0,Y 509.868,Z 268.589,A -85,B 0,C 180,E1 -5519.75,E2 -5519.75} C_VEL
LIN {X 0,Y 510.018,Z 262.8,A -85,B 0,C 180,E1 -5522.796,E2 -5522.796} C_VEL
LIN {X 0,Y 510.194,Z 257.723,A -85,B 0,C 180,E1 -5525.633,E2 -5525.633} C_VEL
LIN {X 0,Y 510.453,Z 253.247,A -85,B 0,C 180,E1 -5528.296,E2 -5528.296} C_VEL
LIN {X 0,Y 510.563,Z 248.46,A -85,B 0,C 180,E1 -5531.355,E2 -5531.355} C_VEL
LIN {X 0,Y 510.257,Z 245.395,A -85,B 0,C 180,E1 -5533.524,E2 -5533.524} C_VEL
LIN {X 0,Y 509.815,Z 242.482,A -85,B 0,C 180,E1 -5535.793,E2 -5535.793} C_VEL
LIN {X 0,Y 509.808,Z 242.483,A -85,B 0,C 180,E1 -5538.567,E2 -5538.567} C_VEL
LIN {X 0,Y 509.826,Z 242.477,A -85,B 0,C 180,E1 -5541.657,E2 -5541.657} C_VEL
LIN {X 0,Y 509.823,Z 242.481,A -85,B 0,C 180,E1 -5544.618,E2 -5544.618} C_VEL
LIN {X 0,Y 509.862,Z 242.47,A -85,B 0,C 180,E1 -5547.478,E2 -5547.478} C_VEL
LIN {X 0,Y 509.858,Z 242.474,A -85,B 0,C 180,E1 -5550.272,E2 -5550.272} C_VEL
LIN {X 0,Y 509.822,Z 242.477,A -85,B 0,C 180,E1 -5552.937,E2 -5552.937} C_VEL
LIN {X 0,Y 509.837,Z 242.473,A -85,B 0,C 180,E1 -5555.569,E2 -5555.569} C_VEL
LIN {X 0,Y 509.819,Z 242.481,A -85,B 0,C 180,E1 -5558.145,E2 -5558.145} C_VEL
LIN {X 0,Y 509.845,Z 242.475,A -85,B 0,C 180,E1 -5560.677,E2 -5560.677} C_VEL
